REGION Network 86: Reset AI_PLC1_Loi_Truyen_Thong từ nút vật lý
   RUNG wire#powerrail
      Contact( "AI_Nut_Reset_Eff" )
      I_Contact( "AI_PLC1_EStop_Latch" )
      I_Contact( "AI_Nut_EStop_Eff" )
      R_Coil( "AI_PLC1_Loi_Truyen_Thong" )
   END_RUNG
   // the same network as SCL:
   IF "AI_Nut_Reset_Eff" AND NOT "AI_PLC1_EStop_Latch" AND NOT "AI_Nut_EStop_Eff" THEN
       "AI_PLC1_Loi_Truyen_Thong" := FALSE;
   END_IF;
END_REGION

REGION Network 87: Reset AI_PID_Bon2_Error từ nút vật lý
   RUNG wire#powerrail
      Contact( "AI_Nut_Reset_Eff" )
      I_Contact( "AI_PLC1_EStop_Latch" )
      I_Contact( "AI_Nut_EStop_Eff" )
      R_Coil( "AI_PID_Bon2_Error" )
   END_RUNG
   // the same network as SCL:
   IF "AI_Nut_Reset_Eff" AND NOT "AI_PLC1_EStop_Latch" AND NOT "AI_Nut_EStop_Eff" THEN
       "AI_PID_Bon2_Error" := FALSE;
   END_IF;
END_REGION

REGION Network 88: Reset AI_PLC1_Loi_Setpoint từ nút vật lý
   RUNG wire#powerrail
      Contact( "AI_Nut_Reset_Eff" )
      I_Contact( "AI_PLC1_EStop_Latch" )
      I_Contact( "AI_Nut_EStop_Eff" )
      R_Coil( "AI_PLC1_Loi_Setpoint" )
   END_RUNG
   // the same network as SCL:
   IF "AI_Nut_Reset_Eff" AND NOT "AI_PLC1_EStop_Latch" AND NOT "AI_Nut_EStop_Eff" THEN
       "AI_PLC1_Loi_Setpoint" := FALSE;
   END_IF;
END_REGION

REGION Network 89: Reset AI_BonChua_Loi_Setpoint từ nút vật lý
   RUNG wire#powerrail
      Contact( "AI_Nut_Reset_Eff" )
      I_Contact( "AI_PLC1_EStop_Latch" )
      I_Contact( "AI_Nut_EStop_Eff" )
      R_Coil( "AI_BonChua_Loi_Setpoint" )
   END_RUNG
   // the same network as SCL:
   IF "AI_Nut_Reset_Eff" AND NOT "AI_PLC1_EStop_Latch" AND NOT "AI_Nut_EStop_Eff" THEN
       "AI_BonChua_Loi_Setpoint" := FALSE;
   END_IF;
END_REGION

REGION Network 90: Reset AI_PLC1_Loi_Tong từ HMI
   RUNG wire#powerrail
      Contact( "AI_HMI_Reset_Alarm" )
      Contact( "AI_HMI_Cho_Phep_Sua_Thong_So" )
      I_Contact( "AI_PLC1_EStop_Latch" )
      I_Contact( "AI_Nut_EStop_Eff" )
      R_Coil( "AI_PLC1_Loi_Tong" )
   END_RUNG
   // the same network as SCL:
   IF "AI_HMI_Reset_Alarm" AND "AI_HMI_Cho_Phep_Sua_Thong_So" AND NOT "AI_PLC1_EStop_Latch" AND NOT "AI_Nut_EStop_Eff" THEN
       "AI_PLC1_Loi_Tong" := FALSE;
   END_IF;
END_REGION

REGION Network 91: Reset AI_PLC1_Loi_Dry_Run từ HMI
   RUNG wire#powerrail
      Contact( "AI_HMI_Reset_Alarm" )
      Contact( "AI_HMI_Cho_Phep_Sua_Thong_So" )
      I_Contact( "AI_PLC1_EStop_Latch" )
      I_Contact( "AI_Nut_EStop_Eff" )
      R_Coil( "AI_PLC1_Loi_Dry_Run" )
   END_RUNG
   // the same network as SCL:
   IF "AI_HMI_Reset_Alarm" AND "AI_HMI_Cho_Phep_Sua_Thong_So" AND NOT "AI_PLC1_EStop_Latch" AND NOT "AI_Nut_EStop_Eff" THEN
       "AI_PLC1_Loi_Dry_Run" := FALSE;
   END_IF;
END_REGION

REGION Network 92: Reset AI_PLC1_Loi_Dosing từ HMI
   RUNG wire#powerrail
      Contact( "AI_HMI_Reset_Alarm" )
      Contact( "AI_HMI_Cho_Phep_Sua_Thong_So" )
      I_Contact( "AI_PLC1_EStop_Latch" )
      I_Contact( "AI_Nut_EStop_Eff" )
      R_Coil( "AI_PLC1_Loi_Dosing" )
   END_RUNG
   // the same network as SCL:
   IF "AI_HMI_Reset_Alarm" AND "AI_HMI_Cho_Phep_Sua_Thong_So" AND NOT "AI_PLC1_EStop_Latch" AND NOT "AI_Nut_EStop_Eff" THEN
       "AI_PLC1_Loi_Dosing" := FALSE;
   END_IF;
END_REGION

REGION Network 93: Reset AI_PLC1_Loi_Truyen_Thong từ HMI
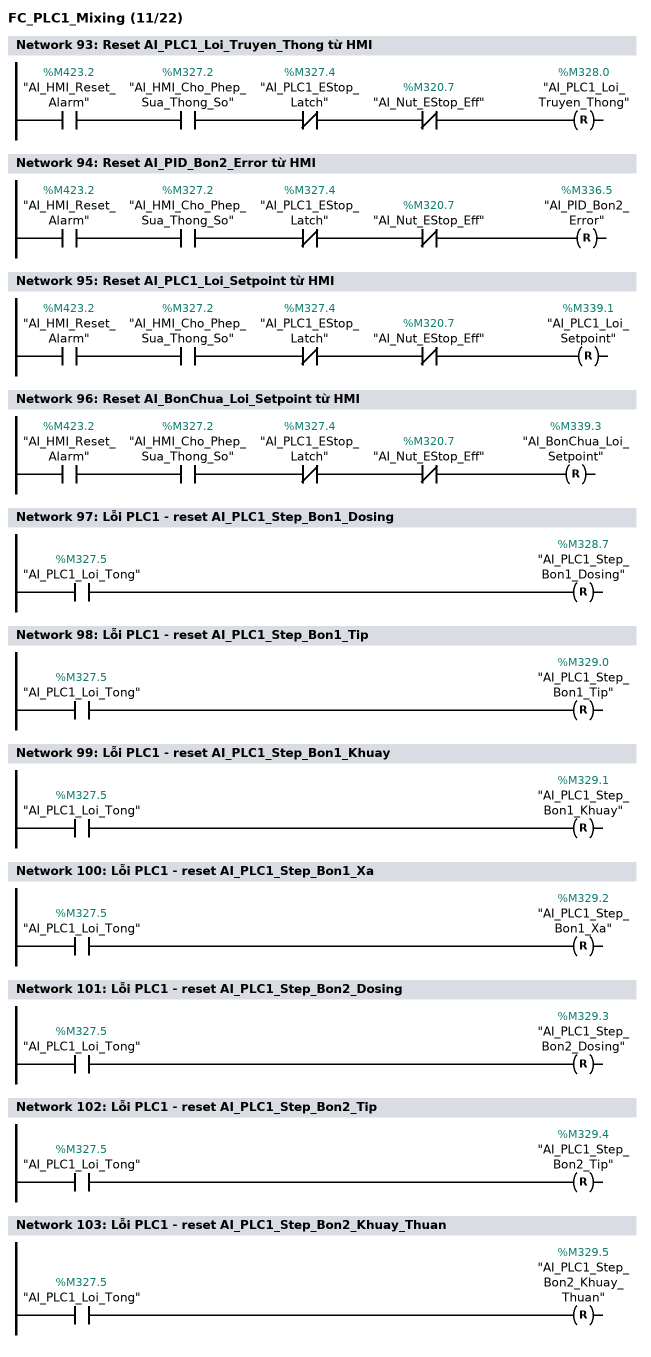
   RUNG wire#powerrail
      Contact( "AI_HMI_Reset_Alarm" )
      Contact( "AI_HMI_Cho_Phep_Sua_Thong_So" )
      I_Contact( "AI_PLC1_EStop_Latch" )
      I_Contact( "AI_Nut_EStop_Eff" )
      R_Coil( "AI_PLC1_Loi_Truyen_Thong" )
   END_RUNG
   // the same network as SCL:
   IF "AI_HMI_Reset_Alarm" AND "AI_HMI_Cho_Phep_Sua_Thong_So" AND NOT "AI_PLC1_EStop_Latch" AND NOT "AI_Nut_EStop_Eff" THEN
       "AI_PLC1_Loi_Truyen_Thong" := FALSE;
   END_IF;
END_REGION

REGION Network 94: Reset AI_PID_Bon2_Error từ HMI
   RUNG wire#powerrail
      Contact( "AI_HMI_Reset_Alarm" )
      Contact( "AI_HMI_Cho_Phep_Sua_Thong_So" )
      I_Contact( "AI_PLC1_EStop_Latch" )
      I_Contact( "AI_Nut_EStop_Eff" )
      R_Coil( "AI_PID_Bon2_Error" )
   END_RUNG
   // the same network as SCL:
   IF "AI_HMI_Reset_Alarm" AND "AI_HMI_Cho_Phep_Sua_Thong_So" AND NOT "AI_PLC1_EStop_Latch" AND NOT "AI_Nut_EStop_Eff" THEN
       "AI_PID_Bon2_Error" := FALSE;
   END_IF;
END_REGION

REGION Network 95: Reset AI_PLC1_Loi_Setpoint từ HMI
   RUNG wire#powerrail
      Contact( "AI_HMI_Reset_Alarm" )
      Contact( "AI_HMI_Cho_Phep_Sua_Thong_So" )
      I_Contact( "AI_PLC1_EStop_Latch" )
      I_Contact( "AI_Nut_EStop_Eff" )
      R_Coil( "AI_PLC1_Loi_Setpoint" )
   END_RUNG
   // the same network as SCL:
   IF "AI_HMI_Reset_Alarm" AND "AI_HMI_Cho_Phep_Sua_Thong_So" AND NOT "AI_PLC1_EStop_Latch" AND NOT "AI_Nut_EStop_Eff" THEN
       "AI_PLC1_Loi_Setpoint" := FALSE;
   END_IF;
END_REGION

REGION Network 96: Reset AI_BonChua_Loi_Setpoint từ HMI
   RUNG wire#powerrail
      Contact( "AI_HMI_Reset_Alarm" )
      Contact( "AI_HMI_Cho_Phep_Sua_Thong_So" )
      I_Contact( "AI_PLC1_EStop_Latch" )
      I_Contact( "AI_Nut_EStop_Eff" )
      R_Coil( "AI_BonChua_Loi_Setpoint" )
   END_RUNG
   // the same network as SCL:
   IF "AI_HMI_Reset_Alarm" AND "AI_HMI_Cho_Phep_Sua_Thong_So" AND NOT "AI_PLC1_EStop_Latch" AND NOT "AI_Nut_EStop_Eff" THEN
       "AI_BonChua_Loi_Setpoint" := FALSE;
   END_IF;
END_REGION

REGION Network 97: Lỗi PLC1 - reset AI_PLC1_Step_Bon1_Dosing
   RUNG wire#powerrail
      Contact( "AI_PLC1_Loi_Tong" )
      R_Coil( "AI_PLC1_Step_Bon1_Dosing" )
   END_RUNG
   // the same network as SCL:
   IF "AI_PLC1_Loi_Tong" THEN "AI_PLC1_Step_Bon1_Dosing" := FALSE; END_IF;
END_REGION

REGION Network 98: Lỗi PLC1 - reset AI_PLC1_Step_Bon1_Tip
   RUNG wire#powerrail
      Contact( "AI_PLC1_Loi_Tong" )
      R_Coil( "AI_PLC1_Step_Bon1_Tip" )
   END_RUNG
   // the same network as SCL:
   IF "AI_PLC1_Loi_Tong" THEN "AI_PLC1_Step_Bon1_Tip" := FALSE; END_IF;
END_REGION

REGION Network 99: Lỗi PLC1 - reset AI_PLC1_Step_Bon1_Khuay
   RUNG wire#powerrail
      Contact( "AI_PLC1_Loi_Tong" )
      R_Coil( "AI_PLC1_Step_Bon1_Khuay" )
   END_RUNG
   // the same network as SCL:
   IF "AI_PLC1_Loi_Tong" THEN "AI_PLC1_Step_Bon1_Khuay" := FALSE; END_IF;
END_REGION

REGION Network 100: Lỗi PLC1 - reset AI_PLC1_Step_Bon1_Xa
   RUNG wire#powerrail
      Contact( "AI_PLC1_Loi_Tong" )
      R_Coil( "AI_PLC1_Step_Bon1_Xa" )
   END_RUNG
   // the same network as SCL:
   IF "AI_PLC1_Loi_Tong" THEN "AI_PLC1_Step_Bon1_Xa" := FALSE; END_IF;
END_REGION

REGION Network 101: Lỗi PLC1 - reset AI_PLC1_Step_Bon2_Dosing
   RUNG wire#powerrail
      Contact( "AI_PLC1_Loi_Tong" )
      R_Coil( "AI_PLC1_Step_Bon2_Dosing" )
   END_RUNG
   // the same network as SCL:
   IF "AI_PLC1_Loi_Tong" THEN "AI_PLC1_Step_Bon2_Dosing" := FALSE; END_IF;
END_REGION

REGION Network 102: Lỗi PLC1 - reset AI_PLC1_Step_Bon2_Tip
   RUNG wire#powerrail
      Contact( "AI_PLC1_Loi_Tong" )
      R_Coil( "AI_PLC1_Step_Bon2_Tip" )
   END_RUNG
   // the same network as SCL:
   IF "AI_PLC1_Loi_Tong" THEN "AI_PLC1_Step_Bon2_Tip" := FALSE; END_IF;
END_REGION

REGION Network 103: Lỗi PLC1 - reset AI_PLC1_Step_Bon2_Khuay_Thuan
   RUNG wire#powerrail
      Contact( "AI_PLC1_Loi_Tong" )
      R_Coil( "AI_PLC1_Step_Bon2_Khuay_Thuan" )
   END_RUNG
   // the same network as SCL:
   IF "AI_PLC1_Loi_Tong" THEN "AI_PLC1_Step_Bon2_Khuay_Thuan" := FALSE; END_IF;
END_REGION

REGION Network 104: Lỗi PLC1 - reset AI_PLC1_Step_Bon2_Khuay_Nghich
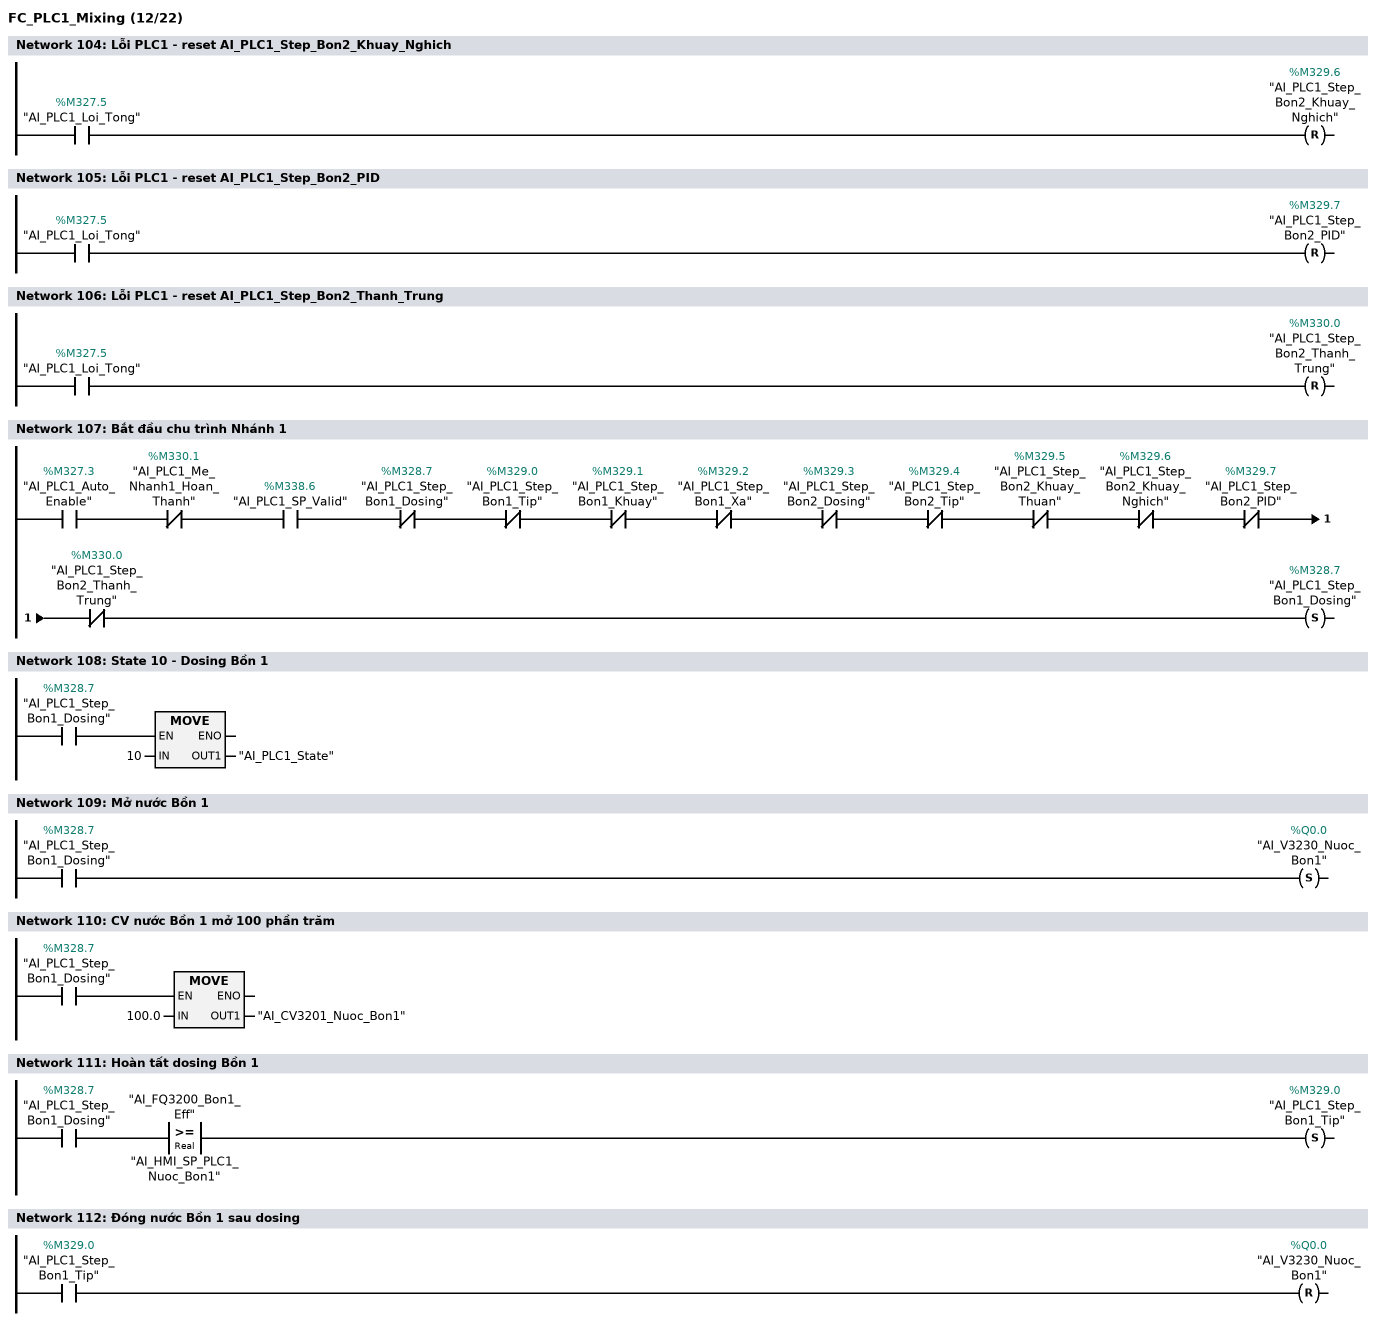
   RUNG wire#powerrail
      Contact( "AI_PLC1_Loi_Tong" )
      R_Coil( "AI_PLC1_Step_Bon2_Khuay_Nghich" )
   END_RUNG
   // the same network as SCL:
   IF "AI_PLC1_Loi_Tong" THEN "AI_PLC1_Step_Bon2_Khuay_Nghich" := FALSE; END_IF;
END_REGION

REGION Network 105: Lỗi PLC1 - reset AI_PLC1_Step_Bon2_PID
   RUNG wire#powerrail
      Contact( "AI_PLC1_Loi_Tong" )
      R_Coil( "AI_PLC1_Step_Bon2_PID" )
   END_RUNG
   // the same network as SCL:
   IF "AI_PLC1_Loi_Tong" THEN "AI_PLC1_Step_Bon2_PID" := FALSE; END_IF;
END_REGION

REGION Network 106: Lỗi PLC1 - reset AI_PLC1_Step_Bon2_Thanh_Trung
   RUNG wire#powerrail
      Contact( "AI_PLC1_Loi_Tong" )
      R_Coil( "AI_PLC1_Step_Bon2_Thanh_Trung" )
   END_RUNG
   // the same network as SCL:
   IF "AI_PLC1_Loi_Tong" THEN "AI_PLC1_Step_Bon2_Thanh_Trung" := FALSE; END_IF;
END_REGION

REGION Network 107: Bắt đầu chu trình Nhánh 1
   RUNG wire#powerrail
      Contact( "AI_PLC1_Auto_Enable" )
      I_Contact( "AI_PLC1_Me_Nhanh1_Hoan_Thanh" )
      Contact( "AI_PLC1_SP_Valid" )
      I_Contact( "AI_PLC1_Step_Bon1_Dosing" )
      I_Contact( "AI_PLC1_Step_Bon1_Tip" )
      I_Contact( "AI_PLC1_Step_Bon1_Khuay" )
      I_Contact( "AI_PLC1_Step_Bon1_Xa" )
      I_Contact( "AI_PLC1_Step_Bon2_Dosing" )
      I_Contact( "AI_PLC1_Step_Bon2_Tip" )
      I_Contact( "AI_PLC1_Step_Bon2_Khuay_Thuan" )
      I_Contact( "AI_PLC1_Step_Bon2_Khuay_Nghich" )
      I_Contact( "AI_PLC1_Step_Bon2_PID" )
      I_Contact( "AI_PLC1_Step_Bon2_Thanh_Trung" )
      S_Coil( "AI_PLC1_Step_Bon1_Dosing" )
   END_RUNG
   // the same network as SCL:
   IF "AI_PLC1_Auto_Enable" AND NOT "AI_PLC1_Me_Nhanh1_Hoan_Thanh" AND "AI_PLC1_SP_Valid" AND NOT "AI_PLC1_Step_Bon1_Dosing" AND NOT "AI_PLC1_Step_Bon1_Tip" AND NOT "AI_PLC1_Step_Bon1_Khuay" AND NOT "AI_PLC1_Step_Bon1_Xa" AND NOT "AI_PLC1_Step_Bon2_Dosing" AND NOT "AI_PLC1_Step_Bon2_Tip" AND NOT "AI_PLC1_Step_Bon2_Khuay_Thuan" AND NOT "AI_PLC1_Step_Bon2_Khuay_Nghich" AND NOT "AI_PLC1_Step_Bon2_PID" AND NOT "AI_PLC1_Step_Bon2_Thanh_Trung" THEN
       "AI_PLC1_Step_Bon1_Dosing" := TRUE;
   END_IF;
END_REGION

REGION Network 108: State 10 - Dosing Bồn 1
   RUNG wire#powerrail
      Contact( "AI_PLC1_Step_Bon1_Dosing" )
      { S7_GenerateENO := "TRUE" } Move(in := 10, out1 => "AI_PLC1_State")
   END_RUNG
   // the same network as SCL:
   IF "AI_PLC1_Step_Bon1_Dosing" THEN "AI_PLC1_State" := 10; END_IF;
END_REGION

REGION Network 109: Mở nước Bồn 1
   RUNG wire#powerrail
      Contact( "AI_PLC1_Step_Bon1_Dosing" )
      S_Coil( "AI_V3230_Nuoc_Bon1" )
   END_RUNG
   // the same network as SCL:
   IF "AI_PLC1_Step_Bon1_Dosing" THEN "AI_V3230_Nuoc_Bon1" := TRUE; END_IF;
END_REGION

REGION Network 110: CV nước Bồn 1 mở 100 phần trăm
   RUNG wire#powerrail
      Contact( "AI_PLC1_Step_Bon1_Dosing" )
      { S7_GenerateENO := "TRUE" } Move(in := 100.0, out1 => "AI_CV3201_Nuoc_Bon1")
   END_RUNG
   // the same network as SCL:
   IF "AI_PLC1_Step_Bon1_Dosing" THEN "AI_CV3201_Nuoc_Bon1" := 100.0; END_IF;
END_REGION

REGION Network 111: Hoàn tất dosing Bồn 1
   RUNG wire#powerrail
      Contact( "AI_PLC1_Step_Bon1_Dosing" )
      { S7_Templates := "SrcType := Real" } GE_Contact(in1 := "AI_FQ3200_Bon1_Eff", in2 := "AI_HMI_SP_PLC1_Nuoc_Bon1")
      S_Coil( "AI_PLC1_Step_Bon1_Tip" )
   END_RUNG
   // the same network as SCL:
   IF "AI_PLC1_Step_Bon1_Dosing" AND ("AI_FQ3200_Bon1_Eff" >= "AI_HMI_SP_PLC1_Nuoc_Bon1") THEN
       "AI_PLC1_Step_Bon1_Tip" := TRUE;
   END_IF;
END_REGION

REGION Network 112: Đóng nước Bồn 1 sau dosing
   RUNG wire#powerrail
      Contact( "AI_PLC1_Step_Bon1_Tip" )
      R_Coil( "AI_V3230_Nuoc_Bon1" )
   END_RUNG
   // the same network as SCL:
   IF "AI_PLC1_Step_Bon1_Tip" THEN "AI_V3230_Nuoc_Bon1" := FALSE; END_IF;
END_REGION

REGION Network 113: Reset bước dosing Bồn 1
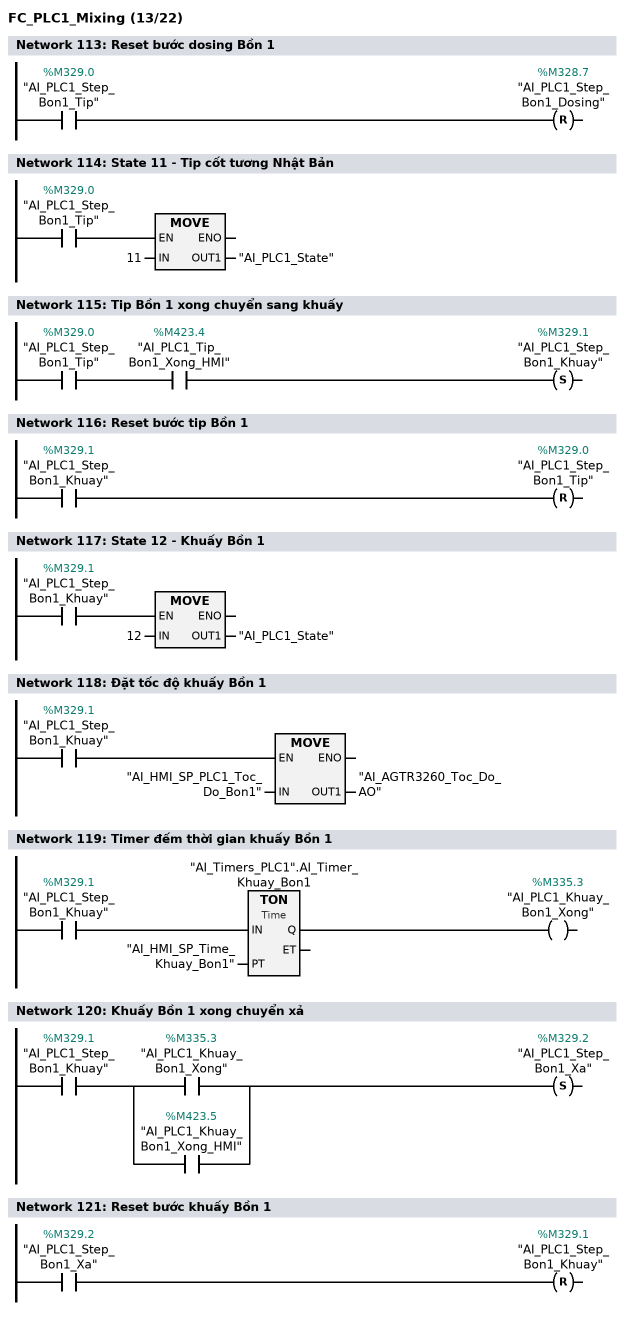
   RUNG wire#powerrail
      Contact( "AI_PLC1_Step_Bon1_Tip" )
      R_Coil( "AI_PLC1_Step_Bon1_Dosing" )
   END_RUNG
   // the same network as SCL:
   IF "AI_PLC1_Step_Bon1_Tip" THEN "AI_PLC1_Step_Bon1_Dosing" := FALSE; END_IF;
END_REGION

REGION Network 114: State 11 - Tip cốt tương Nhật Bản
   RUNG wire#powerrail
      Contact( "AI_PLC1_Step_Bon1_Tip" )
      { S7_GenerateENO := "TRUE" } Move(in := 11, out1 => "AI_PLC1_State")
   END_RUNG
   // the same network as SCL:
   IF "AI_PLC1_Step_Bon1_Tip" THEN "AI_PLC1_State" := 11; END_IF;
END_REGION

REGION Network 115: Tip Bồn 1 xong chuyển sang khuấy
   RUNG wire#powerrail
      Contact( "AI_PLC1_Step_Bon1_Tip" )
      Contact( "AI_PLC1_Tip_Bon1_Xong_HMI" )
      S_Coil( "AI_PLC1_Step_Bon1_Khuay" )
   END_RUNG
   // the same network as SCL:
   IF "AI_PLC1_Step_Bon1_Tip" AND "AI_PLC1_Tip_Bon1_Xong_HMI" THEN "AI_PLC1_Step_Bon1_Khuay" := TRUE; END_IF;
END_REGION

REGION Network 116: Reset bước tip Bồn 1
   RUNG wire#powerrail
      Contact( "AI_PLC1_Step_Bon1_Khuay" )
      R_Coil( "AI_PLC1_Step_Bon1_Tip" )
   END_RUNG
   // the same network as SCL:
   IF "AI_PLC1_Step_Bon1_Khuay" THEN "AI_PLC1_Step_Bon1_Tip" := FALSE; END_IF;
END_REGION

REGION Network 117: State 12 - Khuấy Bồn 1
   RUNG wire#powerrail
      Contact( "AI_PLC1_Step_Bon1_Khuay" )
      { S7_GenerateENO := "TRUE" } Move(in := 12, out1 => "AI_PLC1_State")
   END_RUNG
   // the same network as SCL:
   IF "AI_PLC1_Step_Bon1_Khuay" THEN "AI_PLC1_State" := 12; END_IF;
END_REGION

REGION Network 118: Đặt tốc độ khuấy Bồn 1
   RUNG wire#powerrail
      Contact( "AI_PLC1_Step_Bon1_Khuay" )
      { S7_GenerateENO := "TRUE" } Move(in := "AI_HMI_SP_PLC1_Toc_Do_Bon1", out1 => "AI_AGTR3260_Toc_Do_AO")
   END_RUNG
   // the same network as SCL:
   IF "AI_PLC1_Step_Bon1_Khuay" THEN "AI_AGTR3260_Toc_Do_AO" := "AI_HMI_SP_PLC1_Toc_Do_Bon1"; END_IF;
END_REGION

REGION Network 119: Timer đếm thời gian khuấy Bồn 1
   RUNG wire#powerrail
      Contact( "AI_PLC1_Step_Bon1_Khuay" )
      { S7_Templates := "time_type := Time" } "AI_Timers_PLC1".AI_Timer_Khuay_Bon1.TON(pt := "AI_HMI_SP_Time_Khuay_Bon1", et =>)
      Coil( "AI_PLC1_Khuay_Bon1_Xong" )
   END_RUNG
   // the same network as SCL:
   "AI_Timers_PLC1".AI_Timer_Khuay_Bon1.TON(IN := "AI_PLC1_Step_Bon1_Khuay", PT := "AI_HMI_SP_Time_Khuay_Bon1");
   "AI_PLC1_Khuay_Bon1_Xong" := "AI_Timers_PLC1".AI_Timer_Khuay_Bon1.Q;
END_REGION

REGION Network 120: Khuấy Bồn 1 xong chuyển xả
   RUNG wire#powerrail
      Contact( "AI_PLC1_Step_Bon1_Khuay" )
      wire#w1
      Contact( "AI_PLC1_Khuay_Bon1_Xong" )
      wire#w2
      S_Coil( "AI_PLC1_Step_Bon1_Xa" )
   END_RUNG
   RUNG wire#w1
      Contact( "AI_PLC1_Khuay_Bon1_Xong_HMI" )
   END_RUNG wire#w2
   // the same network as SCL:
   IF "AI_PLC1_Step_Bon1_Khuay" AND ("AI_PLC1_Khuay_Bon1_Xong" OR "AI_PLC1_Khuay_Bon1_Xong_HMI") THEN
       "AI_PLC1_Step_Bon1_Xa" := TRUE;
   END_IF;
END_REGION

REGION Network 121: Reset bước khuấy Bồn 1
   RUNG wire#powerrail
      Contact( "AI_PLC1_Step_Bon1_Xa" )
      R_Coil( "AI_PLC1_Step_Bon1_Khuay" )
   END_RUNG
   // the same network as SCL:
   IF "AI_PLC1_Step_Bon1_Xa" THEN "AI_PLC1_Step_Bon1_Khuay" := FALSE; END_IF;
END_REGION

REGION Network 122: State 15 - Xả Bồn 1 sang Bồn 2
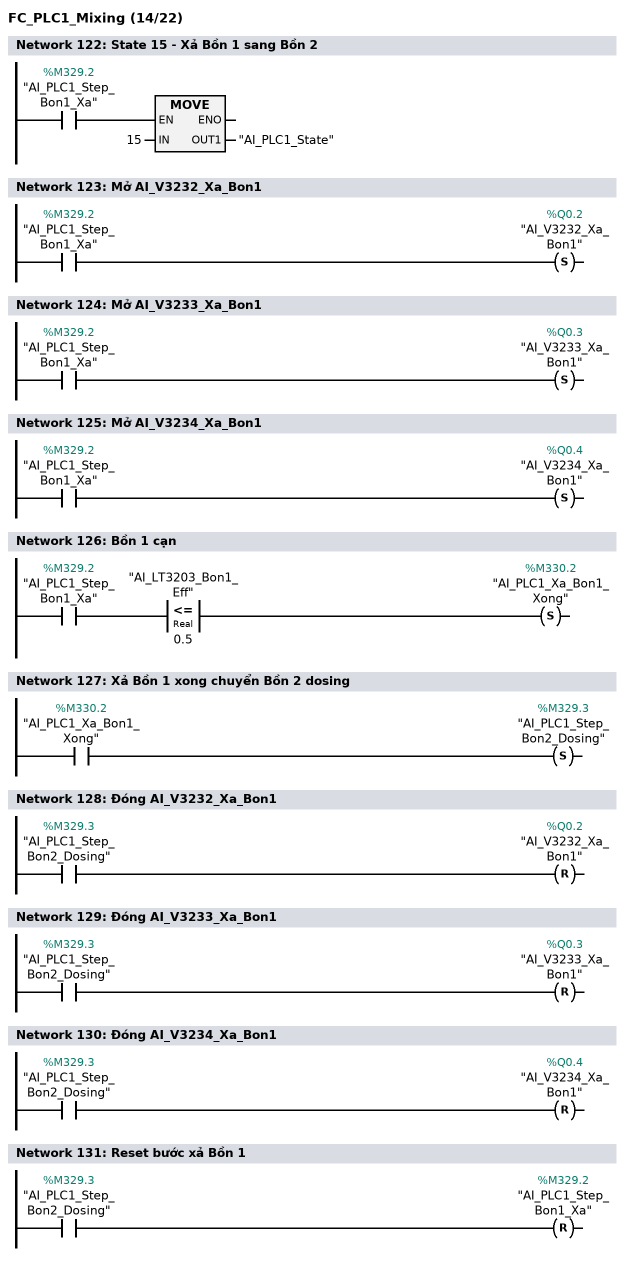
   RUNG wire#powerrail
      Contact( "AI_PLC1_Step_Bon1_Xa" )
      { S7_GenerateENO := "TRUE" } Move(in := 15, out1 => "AI_PLC1_State")
   END_RUNG
   // the same network as SCL:
   IF "AI_PLC1_Step_Bon1_Xa" THEN "AI_PLC1_State" := 15; END_IF;
END_REGION

REGION Network 123: Mở AI_V3232_Xa_Bon1
   RUNG wire#powerrail
      Contact( "AI_PLC1_Step_Bon1_Xa" )
      S_Coil( "AI_V3232_Xa_Bon1" )
   END_RUNG
   // the same network as SCL:
   IF "AI_PLC1_Step_Bon1_Xa" THEN "AI_V3232_Xa_Bon1" := TRUE; END_IF;
END_REGION

REGION Network 124: Mở AI_V3233_Xa_Bon1
   RUNG wire#powerrail
      Contact( "AI_PLC1_Step_Bon1_Xa" )
      S_Coil( "AI_V3233_Xa_Bon1" )
   END_RUNG
   // the same network as SCL:
   IF "AI_PLC1_Step_Bon1_Xa" THEN "AI_V3233_Xa_Bon1" := TRUE; END_IF;
END_REGION

REGION Network 125: Mở AI_V3234_Xa_Bon1
   RUNG wire#powerrail
      Contact( "AI_PLC1_Step_Bon1_Xa" )
      S_Coil( "AI_V3234_Xa_Bon1" )
   END_RUNG
   // the same network as SCL:
   IF "AI_PLC1_Step_Bon1_Xa" THEN "AI_V3234_Xa_Bon1" := TRUE; END_IF;
END_REGION

REGION Network 126: Bồn 1 cạn
   RUNG wire#powerrail
      Contact( "AI_PLC1_Step_Bon1_Xa" )
      { S7_Templates := "SrcType := Real" } LE_Contact(in1 := "AI_LT3203_Bon1_Eff", in2 := 0.5)
      S_Coil( "AI_PLC1_Xa_Bon1_Xong" )
   END_RUNG
   // the same network as SCL:
   IF "AI_PLC1_Step_Bon1_Xa" AND ("AI_LT3203_Bon1_Eff" <= 0.5) THEN "AI_PLC1_Xa_Bon1_Xong" := TRUE; END_IF;
END_REGION

REGION Network 127: Xả Bồn 1 xong chuyển Bồn 2 dosing
   RUNG wire#powerrail
      Contact( "AI_PLC1_Xa_Bon1_Xong" )
      S_Coil( "AI_PLC1_Step_Bon2_Dosing" )
   END_RUNG
   // the same network as SCL:
   IF "AI_PLC1_Xa_Bon1_Xong" THEN "AI_PLC1_Step_Bon2_Dosing" := TRUE; END_IF;
END_REGION

REGION Network 128: Đóng AI_V3232_Xa_Bon1
   RUNG wire#powerrail
      Contact( "AI_PLC1_Step_Bon2_Dosing" )
      R_Coil( "AI_V3232_Xa_Bon1" )
   END_RUNG
   // the same network as SCL:
   IF "AI_PLC1_Step_Bon2_Dosing" THEN "AI_V3232_Xa_Bon1" := FALSE; END_IF;
END_REGION

REGION Network 129: Đóng AI_V3233_Xa_Bon1
   RUNG wire#powerrail
      Contact( "AI_PLC1_Step_Bon2_Dosing" )
      R_Coil( "AI_V3233_Xa_Bon1" )
   END_RUNG
   // the same network as SCL:
   IF "AI_PLC1_Step_Bon2_Dosing" THEN "AI_V3233_Xa_Bon1" := FALSE; END_IF;
END_REGION

REGION Network 130: Đóng AI_V3234_Xa_Bon1
   RUNG wire#powerrail
      Contact( "AI_PLC1_Step_Bon2_Dosing" )
      R_Coil( "AI_V3234_Xa_Bon1" )
   END_RUNG
   // the same network as SCL:
   IF "AI_PLC1_Step_Bon2_Dosing" THEN "AI_V3234_Xa_Bon1" := FALSE; END_IF;
END_REGION

REGION Network 131: Reset bước xả Bồn 1
   RUNG wire#powerrail
      Contact( "AI_PLC1_Step_Bon2_Dosing" )
      R_Coil( "AI_PLC1_Step_Bon1_Xa" )
   END_RUNG
   // the same network as SCL:
   IF "AI_PLC1_Step_Bon2_Dosing" THEN "AI_PLC1_Step_Bon1_Xa" := FALSE; END_IF;
END_REGION

REGION Network 132: State 20 - Dosing Bồn 2
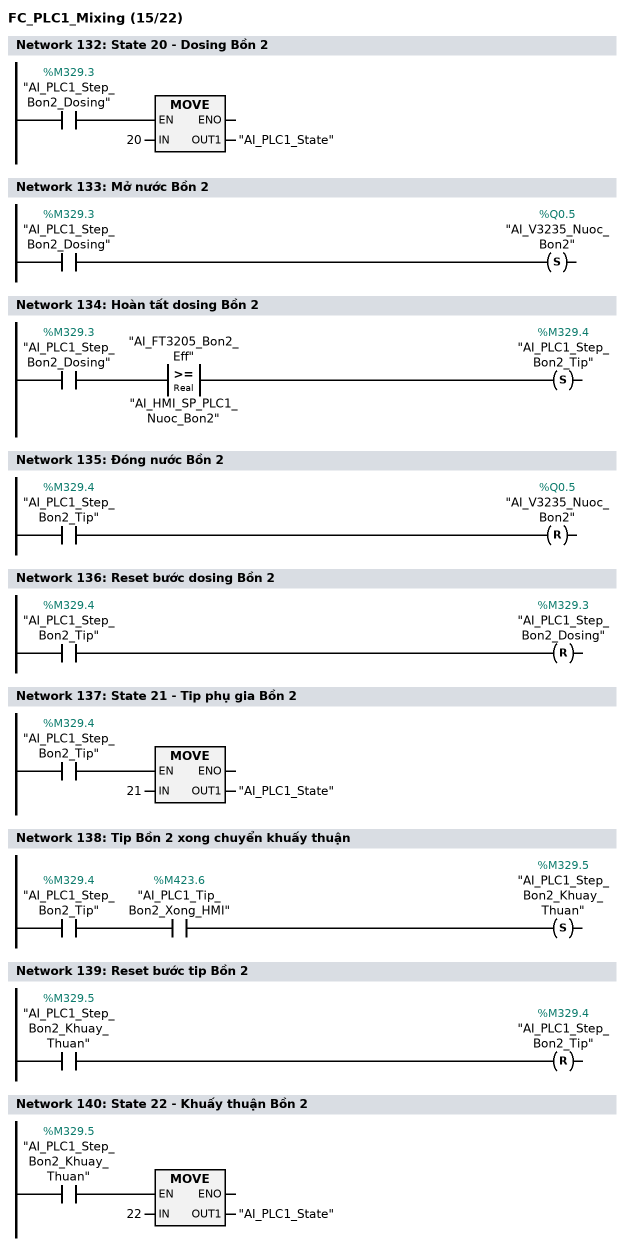
   RUNG wire#powerrail
      Contact( "AI_PLC1_Step_Bon2_Dosing" )
      { S7_GenerateENO := "TRUE" } Move(in := 20, out1 => "AI_PLC1_State")
   END_RUNG
   // the same network as SCL:
   IF "AI_PLC1_Step_Bon2_Dosing" THEN "AI_PLC1_State" := 20; END_IF;
END_REGION

REGION Network 133: Mở nước Bồn 2
   RUNG wire#powerrail
      Contact( "AI_PLC1_Step_Bon2_Dosing" )
      S_Coil( "AI_V3235_Nuoc_Bon2" )
   END_RUNG
   // the same network as SCL:
   IF "AI_PLC1_Step_Bon2_Dosing" THEN "AI_V3235_Nuoc_Bon2" := TRUE; END_IF;
END_REGION

REGION Network 134: Hoàn tất dosing Bồn 2
   RUNG wire#powerrail
      Contact( "AI_PLC1_Step_Bon2_Dosing" )
      { S7_Templates := "SrcType := Real" } GE_Contact(in1 := "AI_FT3205_Bon2_Eff", in2 := "AI_HMI_SP_PLC1_Nuoc_Bon2")
      S_Coil( "AI_PLC1_Step_Bon2_Tip" )
   END_RUNG
   // the same network as SCL:
   IF "AI_PLC1_Step_Bon2_Dosing" AND ("AI_FT3205_Bon2_Eff" >= "AI_HMI_SP_PLC1_Nuoc_Bon2") THEN
       "AI_PLC1_Step_Bon2_Tip" := TRUE;
   END_IF;
END_REGION

REGION Network 135: Đóng nước Bồn 2
   RUNG wire#powerrail
      Contact( "AI_PLC1_Step_Bon2_Tip" )
      R_Coil( "AI_V3235_Nuoc_Bon2" )
   END_RUNG
   // the same network as SCL:
   IF "AI_PLC1_Step_Bon2_Tip" THEN "AI_V3235_Nuoc_Bon2" := FALSE; END_IF;
END_REGION

REGION Network 136: Reset bước dosing Bồn 2
   RUNG wire#powerrail
      Contact( "AI_PLC1_Step_Bon2_Tip" )
      R_Coil( "AI_PLC1_Step_Bon2_Dosing" )
   END_RUNG
   // the same network as SCL:
   IF "AI_PLC1_Step_Bon2_Tip" THEN "AI_PLC1_Step_Bon2_Dosing" := FALSE; END_IF;
END_REGION

REGION Network 137: State 21 - Tip phụ gia Bồn 2
   RUNG wire#powerrail
      Contact( "AI_PLC1_Step_Bon2_Tip" )
      { S7_GenerateENO := "TRUE" } Move(in := 21, out1 => "AI_PLC1_State")
   END_RUNG
   // the same network as SCL:
   IF "AI_PLC1_Step_Bon2_Tip" THEN "AI_PLC1_State" := 21; END_IF;
END_REGION

REGION Network 138: Tip Bồn 2 xong chuyển khuấy thuận
   RUNG wire#powerrail
      Contact( "AI_PLC1_Step_Bon2_Tip" )
      Contact( "AI_PLC1_Tip_Bon2_Xong_HMI" )
      S_Coil( "AI_PLC1_Step_Bon2_Khuay_Thuan" )
   END_RUNG
   // the same network as SCL:
   IF "AI_PLC1_Step_Bon2_Tip" AND "AI_PLC1_Tip_Bon2_Xong_HMI" THEN
       "AI_PLC1_Step_Bon2_Khuay_Thuan" := TRUE;
   END_IF;
END_REGION

REGION Network 139: Reset bước tip Bồn 2
   RUNG wire#powerrail
      Contact( "AI_PLC1_Step_Bon2_Khuay_Thuan" )
      R_Coil( "AI_PLC1_Step_Bon2_Tip" )
   END_RUNG
   // the same network as SCL:
   IF "AI_PLC1_Step_Bon2_Khuay_Thuan" THEN "AI_PLC1_Step_Bon2_Tip" := FALSE; END_IF;
END_REGION

REGION Network 140: State 22 - Khuấy thuận Bồn 2
   RUNG wire#powerrail
      Contact( "AI_PLC1_Step_Bon2_Khuay_Thuan" )
      { S7_GenerateENO := "TRUE" } Move(in := 22, out1 => "AI_PLC1_State")
   END_RUNG
   // the same network as SCL:
   IF "AI_PLC1_Step_Bon2_Khuay_Thuan" THEN "AI_PLC1_State" := 22; END_IF;
END_REGION

REGION Network 141: Tốc độ khuấy thuận Bồn 2
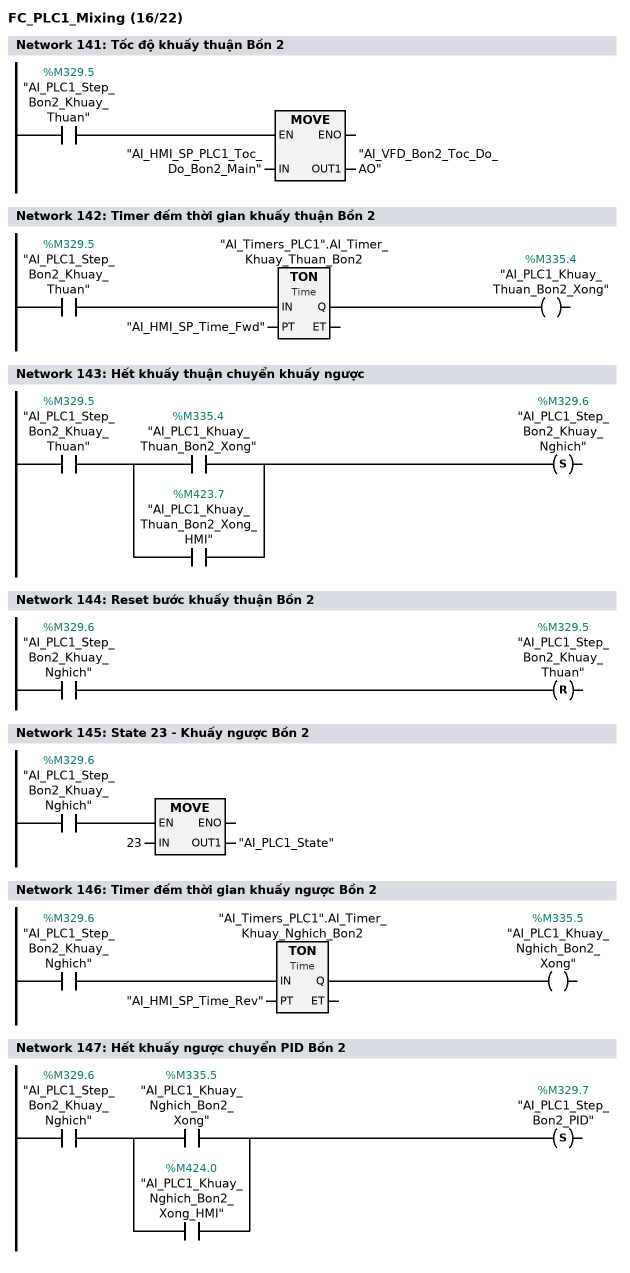
   RUNG wire#powerrail
      Contact( "AI_PLC1_Step_Bon2_Khuay_Thuan" )
      { S7_GenerateENO := "TRUE" } Move(in := "AI_HMI_SP_PLC1_Toc_Do_Bon2_Main", out1 => "AI_VFD_Bon2_Toc_Do_AO")
   END_RUNG
   // the same network as SCL:
   IF "AI_PLC1_Step_Bon2_Khuay_Thuan" THEN
       "AI_VFD_Bon2_Toc_Do_AO" := "AI_HMI_SP_PLC1_Toc_Do_Bon2_Main";
   END_IF;
END_REGION

REGION Network 142: Timer đếm thời gian khuấy thuận Bồn 2
   RUNG wire#powerrail
      Contact( "AI_PLC1_Step_Bon2_Khuay_Thuan" )
      { S7_Templates := "time_type := Time" } "AI_Timers_PLC1".AI_Timer_Khuay_Thuan_Bon2.TON(pt := "AI_HMI_SP_Time_Fwd", et =>)
      Coil( "AI_PLC1_Khuay_Thuan_Bon2_Xong" )
   END_RUNG
   // the same network as SCL:
   "AI_Timers_PLC1".AI_Timer_Khuay_Thuan_Bon2.TON(IN := "AI_PLC1_Step_Bon2_Khuay_Thuan",
                           PT := "AI_HMI_SP_Time_Fwd");
   "AI_PLC1_Khuay_Thuan_Bon2_Xong" := "AI_Timers_PLC1".AI_Timer_Khuay_Thuan_Bon2.Q;
END_REGION

REGION Network 143: Hết khuấy thuận chuyển khuấy ngược
   RUNG wire#powerrail
      Contact( "AI_PLC1_Step_Bon2_Khuay_Thuan" )
      wire#w1
      Contact( "AI_PLC1_Khuay_Thuan_Bon2_Xong" )
      wire#w2
      S_Coil( "AI_PLC1_Step_Bon2_Khuay_Nghich" )
   END_RUNG
   RUNG wire#w1
      Contact( "AI_PLC1_Khuay_Thuan_Bon2_Xong_HMI" )
   END_RUNG wire#w2
   // the same network as SCL:
   IF "AI_PLC1_Step_Bon2_Khuay_Thuan" AND ("AI_PLC1_Khuay_Thuan_Bon2_Xong" OR "AI_PLC1_Khuay_Thuan_Bon2_Xong_HMI") THEN
       "AI_PLC1_Step_Bon2_Khuay_Nghich" := TRUE;
   END_IF;
END_REGION

REGION Network 144: Reset bước khuấy thuận Bồn 2
   RUNG wire#powerrail
      Contact( "AI_PLC1_Step_Bon2_Khuay_Nghich" )
      R_Coil( "AI_PLC1_Step_Bon2_Khuay_Thuan" )
   END_RUNG
   // the same network as SCL:
   IF "AI_PLC1_Step_Bon2_Khuay_Nghich" THEN "AI_PLC1_Step_Bon2_Khuay_Thuan" := FALSE; END_IF;
END_REGION

REGION Network 145: State 23 - Khuấy ngược Bồn 2
   RUNG wire#powerrail
      Contact( "AI_PLC1_Step_Bon2_Khuay_Nghich" )
      { S7_GenerateENO := "TRUE" } Move(in := 23, out1 => "AI_PLC1_State")
   END_RUNG
   // the same network as SCL:
   IF "AI_PLC1_Step_Bon2_Khuay_Nghich" THEN "AI_PLC1_State" := 23; END_IF;
END_REGION

REGION Network 146: Timer đếm thời gian khuấy ngược Bồn 2
   RUNG wire#powerrail
      Contact( "AI_PLC1_Step_Bon2_Khuay_Nghich" )
      { S7_Templates := "time_type := Time" } "AI_Timers_PLC1".AI_Timer_Khuay_Nghich_Bon2.TON(pt := "AI_HMI_SP_Time_Rev", et =>)
      Coil( "AI_PLC1_Khuay_Nghich_Bon2_Xong" )
   END_RUNG
   // the same network as SCL:
   "AI_Timers_PLC1".AI_Timer_Khuay_Nghich_Bon2.TON(IN := "AI_PLC1_Step_Bon2_Khuay_Nghich",
                           PT := "AI_HMI_SP_Time_Rev");
   "AI_PLC1_Khuay_Nghich_Bon2_Xong" := "AI_Timers_PLC1".AI_Timer_Khuay_Nghich_Bon2.Q;
END_REGION

REGION Network 147: Hết khuấy ngược chuyển PID Bồn 2
   RUNG wire#powerrail
      Contact( "AI_PLC1_Step_Bon2_Khuay_Nghich" )
      wire#w1
      Contact( "AI_PLC1_Khuay_Nghich_Bon2_Xong" )
      wire#w2
      S_Coil( "AI_PLC1_Step_Bon2_PID" )
   END_RUNG
   RUNG wire#w1
      Contact( "AI_PLC1_Khuay_Nghich_Bon2_Xong_HMI" )
   END_RUNG wire#w2
   // the same network as SCL:
   IF "AI_PLC1_Step_Bon2_Khuay_Nghich" AND ("AI_PLC1_Khuay_Nghich_Bon2_Xong" OR "AI_PLC1_Khuay_Nghich_Bon2_Xong_HMI") THEN
       "AI_PLC1_Step_Bon2_PID" := TRUE;
   END_IF;
END_REGION

REGION Network 148: Reset bước khuấy ngược Bồn 2
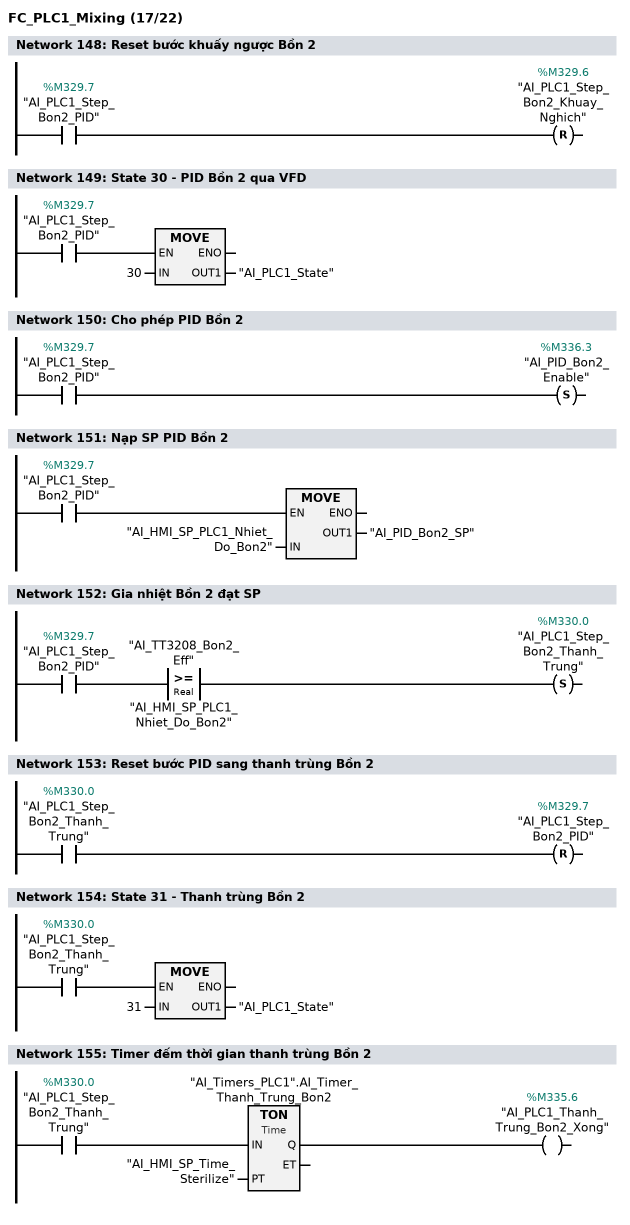
   RUNG wire#powerrail
      Contact( "AI_PLC1_Step_Bon2_PID" )
      R_Coil( "AI_PLC1_Step_Bon2_Khuay_Nghich" )
   END_RUNG
   // the same network as SCL:
   IF "AI_PLC1_Step_Bon2_PID" THEN "AI_PLC1_Step_Bon2_Khuay_Nghich" := FALSE; END_IF;
END_REGION

REGION Network 149: State 30 - PID Bồn 2 qua VFD
   RUNG wire#powerrail
      Contact( "AI_PLC1_Step_Bon2_PID" )
      { S7_GenerateENO := "TRUE" } Move(in := 30, out1 => "AI_PLC1_State")
   END_RUNG
   // the same network as SCL:
   IF "AI_PLC1_Step_Bon2_PID" THEN "AI_PLC1_State" := 30; END_IF;
END_REGION

REGION Network 150: Cho phép PID Bồn 2
   RUNG wire#powerrail
      Contact( "AI_PLC1_Step_Bon2_PID" )
      S_Coil( "AI_PID_Bon2_Enable" )
   END_RUNG
   // the same network as SCL:
   IF "AI_PLC1_Step_Bon2_PID" THEN "AI_PID_Bon2_Enable" := TRUE; END_IF;
END_REGION

REGION Network 151: Nạp SP PID Bồn 2
   RUNG wire#powerrail
      Contact( "AI_PLC1_Step_Bon2_PID" )
      { S7_GenerateENO := "TRUE" } Move(in := "AI_HMI_SP_PLC1_Nhiet_Do_Bon2", out1 => "AI_PID_Bon2_SP")
   END_RUNG
   // the same network as SCL:
   IF "AI_PLC1_Step_Bon2_PID" THEN "AI_PID_Bon2_SP" := "AI_HMI_SP_PLC1_Nhiet_Do_Bon2"; END_IF;
END_REGION

REGION Network 152: Gia nhiệt Bồn 2 đạt SP
   RUNG wire#powerrail
      Contact( "AI_PLC1_Step_Bon2_PID" )
      { S7_Templates := "SrcType := Real" } GE_Contact(in1 := "AI_TT3208_Bon2_Eff", in2 := "AI_HMI_SP_PLC1_Nhiet_Do_Bon2")
      S_Coil( "AI_PLC1_Step_Bon2_Thanh_Trung" )
   END_RUNG
   // the same network as SCL:
   IF "AI_PLC1_Step_Bon2_PID" AND ("AI_TT3208_Bon2_Eff" >= "AI_HMI_SP_PLC1_Nhiet_Do_Bon2") THEN
       "AI_PLC1_Step_Bon2_Thanh_Trung" := TRUE;
   END_IF;
END_REGION

REGION Network 153: Reset bước PID sang thanh trùng Bồn 2
   RUNG wire#powerrail
      Contact( "AI_PLC1_Step_Bon2_Thanh_Trung" )
      R_Coil( "AI_PLC1_Step_Bon2_PID" )
   END_RUNG
   // the same network as SCL:
   IF "AI_PLC1_Step_Bon2_Thanh_Trung" THEN "AI_PLC1_Step_Bon2_PID" := FALSE; END_IF;
END_REGION

REGION Network 154: State 31 - Thanh trùng Bồn 2
   RUNG wire#powerrail
      Contact( "AI_PLC1_Step_Bon2_Thanh_Trung" )
      { S7_GenerateENO := "TRUE" } Move(in := 31, out1 => "AI_PLC1_State")
   END_RUNG
   // the same network as SCL:
   IF "AI_PLC1_Step_Bon2_Thanh_Trung" THEN "AI_PLC1_State" := 31; END_IF;
END_REGION

REGION Network 155: Timer đếm thời gian thanh trùng Bồn 2
   RUNG wire#powerrail
      Contact( "AI_PLC1_Step_Bon2_Thanh_Trung" )
      { S7_Templates := "time_type := Time" } "AI_Timers_PLC1".AI_Timer_Thanh_Trung_Bon2.TON(pt := "AI_HMI_SP_Time_Sterilize", et =>)
      Coil( "AI_PLC1_Thanh_Trung_Bon2_Xong" )
   END_RUNG
   // the same network as SCL:
   "AI_Timers_PLC1".AI_Timer_Thanh_Trung_Bon2.TON(IN := "AI_PLC1_Step_Bon2_Thanh_Trung",
                           PT := "AI_HMI_SP_Time_Sterilize");
   "AI_PLC1_Thanh_Trung_Bon2_Xong" := "AI_Timers_PLC1".AI_Timer_Thanh_Trung_Bon2.Q;
END_REGION

REGION Network 156: Thanh trùng Bồn 2 xong
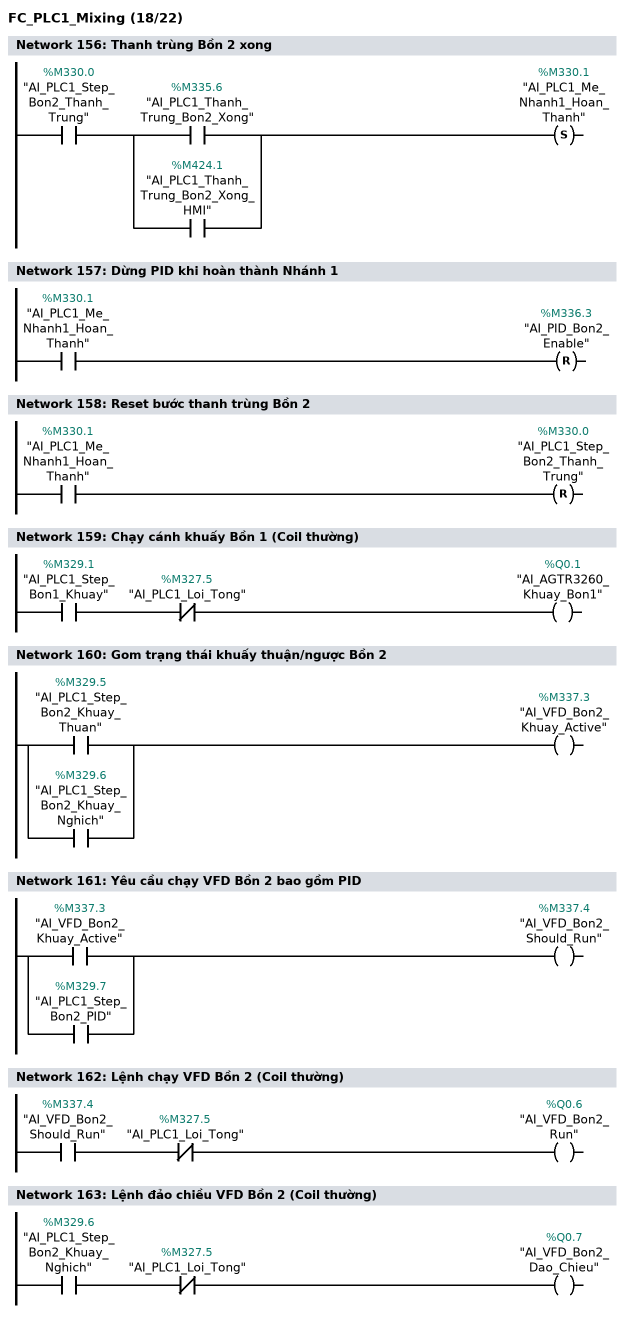
   RUNG wire#powerrail
      Contact( "AI_PLC1_Step_Bon2_Thanh_Trung" )
      wire#w1
      Contact( "AI_PLC1_Thanh_Trung_Bon2_Xong" )
      wire#w2
      S_Coil( "AI_PLC1_Me_Nhanh1_Hoan_Thanh" )
   END_RUNG
   RUNG wire#w1
      Contact( "AI_PLC1_Thanh_Trung_Bon2_Xong_HMI" )
   END_RUNG wire#w2
   // the same network as SCL:
   IF "AI_PLC1_Step_Bon2_Thanh_Trung" AND ("AI_PLC1_Thanh_Trung_Bon2_Xong" OR "AI_PLC1_Thanh_Trung_Bon2_Xong_HMI") THEN
       "AI_PLC1_Me_Nhanh1_Hoan_Thanh" := TRUE;
   END_IF;
END_REGION

REGION Network 157: Dừng PID khi hoàn thành Nhánh 1
   RUNG wire#powerrail
      Contact( "AI_PLC1_Me_Nhanh1_Hoan_Thanh" )
      R_Coil( "AI_PID_Bon2_Enable" )
   END_RUNG
   // the same network as SCL:
   IF "AI_PLC1_Me_Nhanh1_Hoan_Thanh" THEN "AI_PID_Bon2_Enable" := FALSE; END_IF;
END_REGION

REGION Network 158: Reset bước thanh trùng Bồn 2
   RUNG wire#powerrail
      Contact( "AI_PLC1_Me_Nhanh1_Hoan_Thanh" )
      R_Coil( "AI_PLC1_Step_Bon2_Thanh_Trung" )
   END_RUNG
   // the same network as SCL:
   IF "AI_PLC1_Me_Nhanh1_Hoan_Thanh" THEN "AI_PLC1_Step_Bon2_Thanh_Trung" := FALSE; END_IF;
END_REGION

REGION Network 159: Chạy cánh khuấy Bồn 1 (Coil thường)
   RUNG wire#powerrail
      Contact( "AI_PLC1_Step_Bon1_Khuay" )
      I_Contact( "AI_PLC1_Loi_Tong" )
      Coil( "AI_AGTR3260_Khuay_Bon1" )
   END_RUNG
   // the same network as SCL:
   "AI_AGTR3260_Khuay_Bon1" := "AI_PLC1_Step_Bon1_Khuay" AND NOT "AI_PLC1_Loi_Tong";
END_REGION

REGION Network 160: Gom trạng thái khuấy thuận/ngược Bồn 2
   RUNG wire#powerrail
      Contact( "AI_PLC1_Step_Bon2_Khuay_Thuan" )
      wire#w1
      Coil( "AI_VFD_Bon2_Khuay_Active" )
   END_RUNG
   RUNG wire#powerrail
      Contact( "AI_PLC1_Step_Bon2_Khuay_Nghich" )
   END_RUNG wire#w1
   // the same network as SCL:
   "AI_VFD_Bon2_Khuay_Active" := "AI_PLC1_Step_Bon2_Khuay_Thuan" OR "AI_PLC1_Step_Bon2_Khuay_Nghich";
END_REGION

REGION Network 161: Yêu cầu chạy VFD Bồn 2 bao gồm PID
   RUNG wire#powerrail
      Contact( "AI_VFD_Bon2_Khuay_Active" )
      wire#w1
      Coil( "AI_VFD_Bon2_Should_Run" )
   END_RUNG
   RUNG wire#powerrail
      Contact( "AI_PLC1_Step_Bon2_PID" )
   END_RUNG wire#w1
   // the same network as SCL:
   "AI_VFD_Bon2_Should_Run" := "AI_VFD_Bon2_Khuay_Active" OR "AI_PLC1_Step_Bon2_PID";
END_REGION

REGION Network 162: Lệnh chạy VFD Bồn 2 (Coil thường)
   RUNG wire#powerrail
      Contact( "AI_VFD_Bon2_Should_Run" )
      I_Contact( "AI_PLC1_Loi_Tong" )
      Coil( "AI_VFD_Bon2_Run" )
   END_RUNG
   // the same network as SCL:
   "AI_VFD_Bon2_Run" := "AI_VFD_Bon2_Should_Run" AND NOT "AI_PLC1_Loi_Tong";
END_REGION

REGION Network 163: Lệnh đảo chiều VFD Bồn 2 (Coil thường)
   RUNG wire#powerrail
      Contact( "AI_PLC1_Step_Bon2_Khuay_Nghich" )
      I_Contact( "AI_PLC1_Loi_Tong" )
      Coil( "AI_VFD_Bon2_Dao_Chieu" )
   END_RUNG
   // the same network as SCL:
   "AI_VFD_Bon2_Dao_Chieu" := "AI_PLC1_Step_Bon2_Khuay_Nghich" AND NOT "AI_PLC1_Loi_Tong";
END_REGION

REGION Network 164: Reset CV nước Bồn 1 khi không dosing
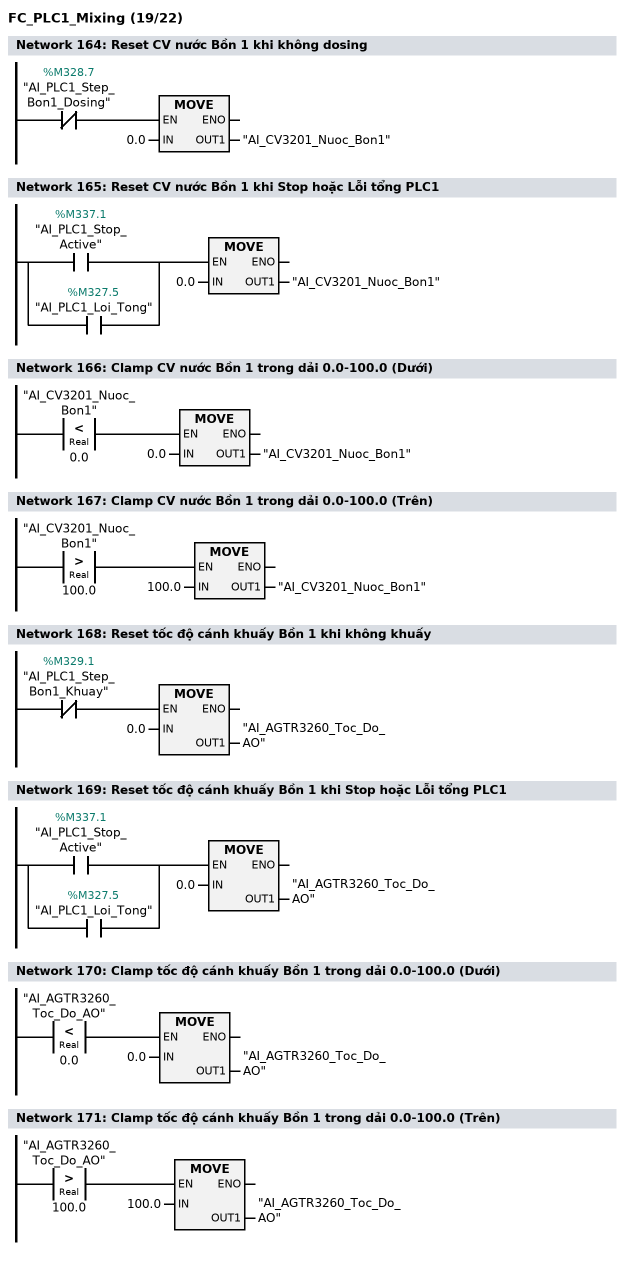
   RUNG wire#powerrail
      I_Contact( "AI_PLC1_Step_Bon1_Dosing" )
      { S7_GenerateENO := "TRUE" } Move(in := 0.0, out1 => "AI_CV3201_Nuoc_Bon1")
   END_RUNG
   // the same network as SCL:
   IF NOT "AI_PLC1_Step_Bon1_Dosing" THEN "AI_CV3201_Nuoc_Bon1" := 0.0; END_IF;
END_REGION

REGION Network 165: Reset CV nước Bồn 1 khi Stop hoặc Lỗi tổng PLC1
   RUNG wire#powerrail
      Contact( "AI_PLC1_Stop_Active" )
      wire#w1
      { S7_GenerateENO := "TRUE" } Move(in := 0.0, out1 => "AI_CV3201_Nuoc_Bon1")
   END_RUNG
   RUNG wire#powerrail
      Contact( "AI_PLC1_Loi_Tong" )
   END_RUNG wire#w1
   // the same network as SCL:
   IF "AI_PLC1_Stop_Active" OR "AI_PLC1_Loi_Tong" THEN "AI_CV3201_Nuoc_Bon1" := 0.0; END_IF;
END_REGION

REGION Network 166: Clamp CV nước Bồn 1 trong dải 0.0-100.0 (Dưới)
   RUNG wire#powerrail
      { S7_Templates := "SrcType := Real" } LT_Contact(in1 := "AI_CV3201_Nuoc_Bon1", in2 := 0.0)
      { S7_GenerateENO := "TRUE" } Move(in := 0.0, out1 => "AI_CV3201_Nuoc_Bon1")
   END_RUNG
   // the same network as SCL:
   IF "AI_CV3201_Nuoc_Bon1" < 0.0 THEN "AI_CV3201_Nuoc_Bon1" := 0.0; END_IF;
END_REGION

REGION Network 167: Clamp CV nước Bồn 1 trong dải 0.0-100.0 (Trên)
   RUNG wire#powerrail
      { S7_Templates := "SrcType := Real" } GT_Contact(in1 := "AI_CV3201_Nuoc_Bon1", in2 := 100.0)
      { S7_GenerateENO := "TRUE" } Move(in := 100.0, out1 => "AI_CV3201_Nuoc_Bon1")
   END_RUNG
   // the same network as SCL:
   IF "AI_CV3201_Nuoc_Bon1" > 100.0 THEN "AI_CV3201_Nuoc_Bon1" := 100.0; END_IF;
END_REGION

REGION Network 168: Reset tốc độ cánh khuấy Bồn 1 khi không khuấy
   RUNG wire#powerrail
      I_Contact( "AI_PLC1_Step_Bon1_Khuay" )
      { S7_GenerateENO := "TRUE" } Move(in := 0.0, out1 => "AI_AGTR3260_Toc_Do_AO")
   END_RUNG
   // the same network as SCL:
   IF NOT "AI_PLC1_Step_Bon1_Khuay" THEN "AI_AGTR3260_Toc_Do_AO" := 0.0; END_IF;
END_REGION

REGION Network 169: Reset tốc độ cánh khuấy Bồn 1 khi Stop hoặc Lỗi tổng PLC1
   RUNG wire#powerrail
      Contact( "AI_PLC1_Stop_Active" )
      wire#w1
      { S7_GenerateENO := "TRUE" } Move(in := 0.0, out1 => "AI_AGTR3260_Toc_Do_AO")
   END_RUNG
   RUNG wire#powerrail
      Contact( "AI_PLC1_Loi_Tong" )
   END_RUNG wire#w1
   // the same network as SCL:
   IF "AI_PLC1_Stop_Active" OR "AI_PLC1_Loi_Tong" THEN "AI_AGTR3260_Toc_Do_AO" := 0.0; END_IF;
END_REGION

REGION Network 170: Clamp tốc độ cánh khuấy Bồn 1 trong dải 0.0-100.0 (Dưới)
   RUNG wire#powerrail
      { S7_Templates := "SrcType := Real" } LT_Contact(in1 := "AI_AGTR3260_Toc_Do_AO", in2 := 0.0)
      { S7_GenerateENO := "TRUE" } Move(in := 0.0, out1 => "AI_AGTR3260_Toc_Do_AO")
   END_RUNG
   // the same network as SCL:
   IF "AI_AGTR3260_Toc_Do_AO" < 0.0 THEN "AI_AGTR3260_Toc_Do_AO" := 0.0; END_IF;
END_REGION

REGION Network 171: Clamp tốc độ cánh khuấy Bồn 1 trong dải 0.0-100.0 (Trên)
   RUNG wire#powerrail
      { S7_Templates := "SrcType := Real" } GT_Contact(in1 := "AI_AGTR3260_Toc_Do_AO", in2 := 100.0)
      { S7_GenerateENO := "TRUE" } Move(in := 100.0, out1 => "AI_AGTR3260_Toc_Do_AO")
   END_RUNG
   // the same network as SCL:
   IF "AI_AGTR3260_Toc_Do_AO" > 100.0 THEN "AI_AGTR3260_Toc_Do_AO" := 100.0; END_IF;
END_REGION

REGION Network 172: Reset CV hơi Bồn 2 khi không chạy PID
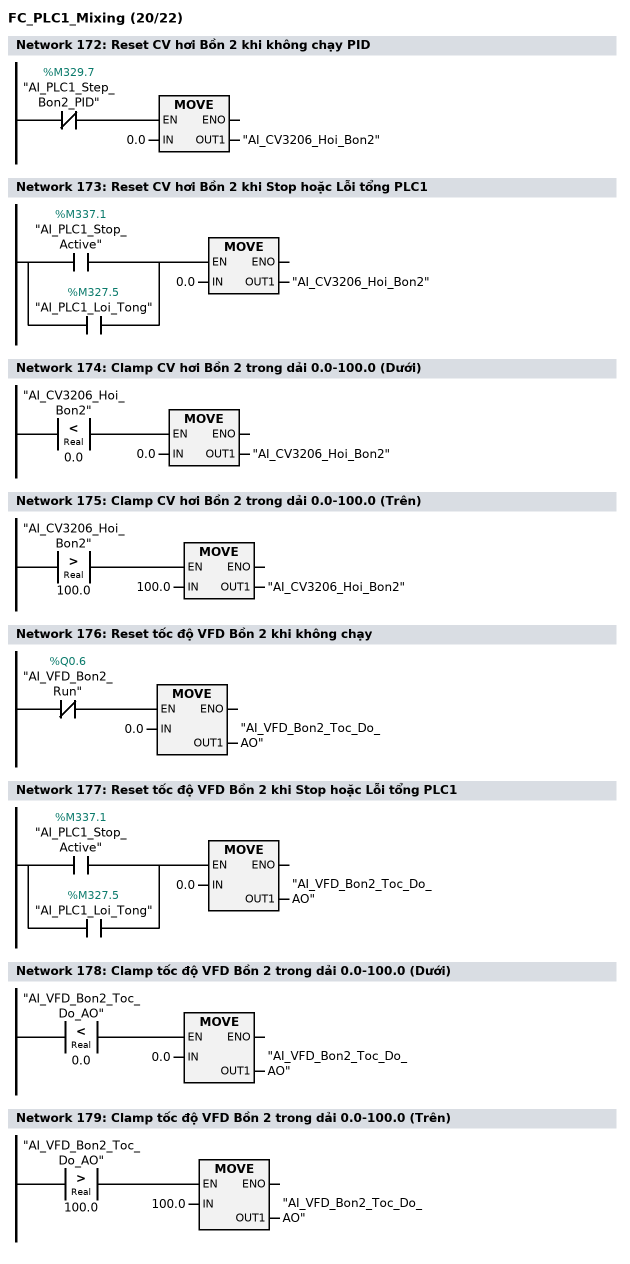
   RUNG wire#powerrail
      I_Contact( "AI_PLC1_Step_Bon2_PID" )
      { S7_GenerateENO := "TRUE" } Move(in := 0.0, out1 => "AI_CV3206_Hoi_Bon2")
   END_RUNG
   // the same network as SCL:
   IF NOT "AI_PLC1_Step_Bon2_PID" THEN "AI_CV3206_Hoi_Bon2" := 0.0; END_IF;
END_REGION

REGION Network 173: Reset CV hơi Bồn 2 khi Stop hoặc Lỗi tổng PLC1
   RUNG wire#powerrail
      Contact( "AI_PLC1_Stop_Active" )
      wire#w1
      { S7_GenerateENO := "TRUE" } Move(in := 0.0, out1 => "AI_CV3206_Hoi_Bon2")
   END_RUNG
   RUNG wire#powerrail
      Contact( "AI_PLC1_Loi_Tong" )
   END_RUNG wire#w1
   // the same network as SCL:
   IF "AI_PLC1_Stop_Active" OR "AI_PLC1_Loi_Tong" THEN "AI_CV3206_Hoi_Bon2" := 0.0; END_IF;
END_REGION

REGION Network 174: Clamp CV hơi Bồn 2 trong dải 0.0-100.0 (Dưới)
   RUNG wire#powerrail
      { S7_Templates := "SrcType := Real" } LT_Contact(in1 := "AI_CV3206_Hoi_Bon2", in2 := 0.0)
      { S7_GenerateENO := "TRUE" } Move(in := 0.0, out1 => "AI_CV3206_Hoi_Bon2")
   END_RUNG
   // the same network as SCL:
   IF "AI_CV3206_Hoi_Bon2" < 0.0 THEN "AI_CV3206_Hoi_Bon2" := 0.0; END_IF;
END_REGION

REGION Network 175: Clamp CV hơi Bồn 2 trong dải 0.0-100.0 (Trên)
   RUNG wire#powerrail
      { S7_Templates := "SrcType := Real" } GT_Contact(in1 := "AI_CV3206_Hoi_Bon2", in2 := 100.0)
      { S7_GenerateENO := "TRUE" } Move(in := 100.0, out1 => "AI_CV3206_Hoi_Bon2")
   END_RUNG
   // the same network as SCL:
   IF "AI_CV3206_Hoi_Bon2" > 100.0 THEN "AI_CV3206_Hoi_Bon2" := 100.0; END_IF;
END_REGION

REGION Network 176: Reset tốc độ VFD Bồn 2 khi không chạy
   RUNG wire#powerrail
      I_Contact( "AI_VFD_Bon2_Run" )
      { S7_GenerateENO := "TRUE" } Move(in := 0.0, out1 => "AI_VFD_Bon2_Toc_Do_AO")
   END_RUNG
   // the same network as SCL:
   IF NOT "AI_VFD_Bon2_Run" THEN "AI_VFD_Bon2_Toc_Do_AO" := 0.0; END_IF;
END_REGION

REGION Network 177: Reset tốc độ VFD Bồn 2 khi Stop hoặc Lỗi tổng PLC1
   RUNG wire#powerrail
      Contact( "AI_PLC1_Stop_Active" )
      wire#w1
      { S7_GenerateENO := "TRUE" } Move(in := 0.0, out1 => "AI_VFD_Bon2_Toc_Do_AO")
   END_RUNG
   RUNG wire#powerrail
      Contact( "AI_PLC1_Loi_Tong" )
   END_RUNG wire#w1
   // the same network as SCL:
   IF "AI_PLC1_Stop_Active" OR "AI_PLC1_Loi_Tong" THEN "AI_VFD_Bon2_Toc_Do_AO" := 0.0; END_IF;
END_REGION

REGION Network 178: Clamp tốc độ VFD Bồn 2 trong dải 0.0-100.0 (Dưới)
   RUNG wire#powerrail
      { S7_Templates := "SrcType := Real" } LT_Contact(in1 := "AI_VFD_Bon2_Toc_Do_AO", in2 := 0.0)
      { S7_GenerateENO := "TRUE" } Move(in := 0.0, out1 => "AI_VFD_Bon2_Toc_Do_AO")
   END_RUNG
   // the same network as SCL:
   IF "AI_VFD_Bon2_Toc_Do_AO" < 0.0 THEN "AI_VFD_Bon2_Toc_Do_AO" := 0.0; END_IF;
END_REGION

REGION Network 179: Clamp tốc độ VFD Bồn 2 trong dải 0.0-100.0 (Trên)
   RUNG wire#powerrail
      { S7_Templates := "SrcType := Real" } GT_Contact(in1 := "AI_VFD_Bon2_Toc_Do_AO", in2 := 100.0)
      { S7_GenerateENO := "TRUE" } Move(in := 100.0, out1 => "AI_VFD_Bon2_Toc_Do_AO")
   END_RUNG
   // the same network as SCL:
   IF "AI_VFD_Bon2_Toc_Do_AO" > 100.0 THEN "AI_VFD_Bon2_Toc_Do_AO" := 100.0; END_IF;
END_REGION

REGION Network 180: VFD Bon 2 Freq Scale: Speed SP x 5.0
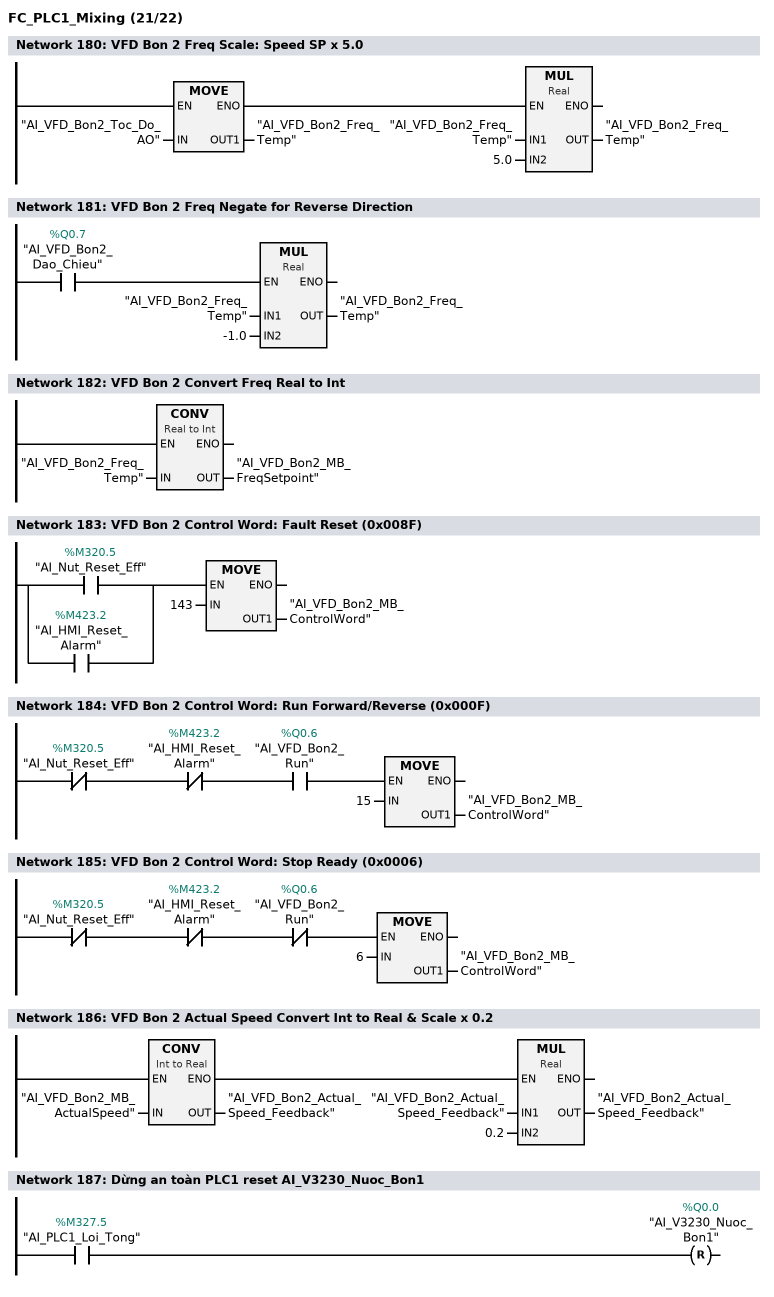
   RUNG wire#powerrail
      { S7_GenerateENO := "TRUE" } Move(in := "AI_VFD_Bon2_Toc_Do_AO", out1 => "AI_VFD_Bon2_Freq_Temp")
      { S7_Templates := "SrcType := Real"; S7_GenerateENO := "TRUE" } Mul(in1 := "AI_VFD_Bon2_Freq_Temp", in2 := 5.0, out => "AI_VFD_Bon2_Freq_Temp")
   END_RUNG
   // the same network as SCL:
   // ENO of a box is taken as its EN; it also drops when the box reports an error
   "AI_VFD_Bon2_Freq_Temp" := "AI_VFD_Bon2_Toc_Do_AO";
   "AI_VFD_Bon2_Freq_Temp" := "AI_VFD_Bon2_Freq_Temp" * 5.0;
END_REGION

REGION Network 181: VFD Bon 2 Freq Negate for Reverse Direction
   RUNG wire#powerrail
      Contact( "AI_VFD_Bon2_Dao_Chieu" )
      { S7_Templates := "SrcType := Real"; S7_GenerateENO := "TRUE" } Mul(in1 := "AI_VFD_Bon2_Freq_Temp", in2 := -1.0, out => "AI_VFD_Bon2_Freq_Temp")
   END_RUNG
   // the same network as SCL:
   IF "AI_VFD_Bon2_Dao_Chieu" THEN "AI_VFD_Bon2_Freq_Temp" := "AI_VFD_Bon2_Freq_Temp" * (-1.0); END_IF;
END_REGION

REGION Network 182: VFD Bon 2 Convert Freq Real to Int
   RUNG wire#powerrail
      { S7_Templates := "[SrcType := Real, DestType := Int]"; S7_GenerateENO := "TRUE" } Convert(in := "AI_VFD_Bon2_Freq_Temp", out => "AI_VFD_Bon2_MB_FreqSetpoint")
   END_RUNG
   // the same network as SCL:
   "AI_VFD_Bon2_MB_FreqSetpoint" := REAL_TO_INT("AI_VFD_Bon2_Freq_Temp");
END_REGION

REGION Network 183: VFD Bon 2 Control Word: Fault Reset (0x008F)
   RUNG wire#powerrail
      Contact( "AI_Nut_Reset_Eff" )
      wire#w1
      { S7_GenerateENO := "TRUE" } Move(in := 143, out1 => "AI_VFD_Bon2_MB_ControlWord")
   END_RUNG
   RUNG wire#powerrail
      Contact( "AI_HMI_Reset_Alarm" )
   END_RUNG wire#w1
   // the same network as SCL:
   IF "AI_Nut_Reset_Eff" OR "AI_HMI_Reset_Alarm" THEN "AI_VFD_Bon2_MB_ControlWord" := 143; END_IF;
END_REGION

REGION Network 184: VFD Bon 2 Control Word: Run Forward/Reverse (0x000F)
   RUNG wire#powerrail
      I_Contact( "AI_Nut_Reset_Eff" )
      I_Contact( "AI_HMI_Reset_Alarm" )
      Contact( "AI_VFD_Bon2_Run" )
      { S7_GenerateENO := "TRUE" } Move(in := 15, out1 => "AI_VFD_Bon2_MB_ControlWord")
   END_RUNG
   // the same network as SCL:
   IF NOT "AI_Nut_Reset_Eff" AND NOT "AI_HMI_Reset_Alarm" AND "AI_VFD_Bon2_Run" THEN
       "AI_VFD_Bon2_MB_ControlWord" := 15;
   END_IF;
END_REGION

REGION Network 185: VFD Bon 2 Control Word: Stop Ready (0x0006)
   RUNG wire#powerrail
      I_Contact( "AI_Nut_Reset_Eff" )
      I_Contact( "AI_HMI_Reset_Alarm" )
      I_Contact( "AI_VFD_Bon2_Run" )
      { S7_GenerateENO := "TRUE" } Move(in := 6, out1 => "AI_VFD_Bon2_MB_ControlWord")
   END_RUNG
   // the same network as SCL:
   IF NOT "AI_Nut_Reset_Eff" AND NOT "AI_HMI_Reset_Alarm" AND NOT "AI_VFD_Bon2_Run" THEN
       "AI_VFD_Bon2_MB_ControlWord" := 6;
   END_IF;
END_REGION

REGION Network 186: VFD Bon 2 Actual Speed Convert Int to Real & Scale x 0.2
   RUNG wire#powerrail
      { S7_Templates := "[SrcType := Int, DestType := Real]"; S7_GenerateENO := "TRUE" } Convert(in := "AI_VFD_Bon2_MB_ActualSpeed", out => "AI_VFD_Bon2_Actual_Speed_Feedback")
      { S7_Templates := "SrcType := Real"; S7_GenerateENO := "TRUE" } Mul(in1 := "AI_VFD_Bon2_Actual_Speed_Feedback", in2 := 0.2, out => "AI_VFD_Bon2_Actual_Speed_Feedback")
   END_RUNG
   // the same network as SCL:
   // ENO of a box is taken as its EN; it also drops when the box reports an error
   "AI_VFD_Bon2_Actual_Speed_Feedback" := INT_TO_REAL("AI_VFD_Bon2_MB_ActualSpeed");
   "AI_VFD_Bon2_Actual_Speed_Feedback" := "AI_VFD_Bon2_Actual_Speed_Feedback" * 0.2;
END_REGION

REGION Network 187: Dừng an toàn PLC1 reset AI_V3230_Nuoc_Bon1
   RUNG wire#powerrail
      Contact( "AI_PLC1_Loi_Tong" )
      R_Coil( "AI_V3230_Nuoc_Bon1" )
   END_RUNG
   // the same network as SCL:
   IF "AI_PLC1_Loi_Tong" THEN "AI_V3230_Nuoc_Bon1" := FALSE; END_IF;
END_REGION

REGION Network 188: Dừng an toàn PLC1 reset AI_V3232_Xa_Bon1
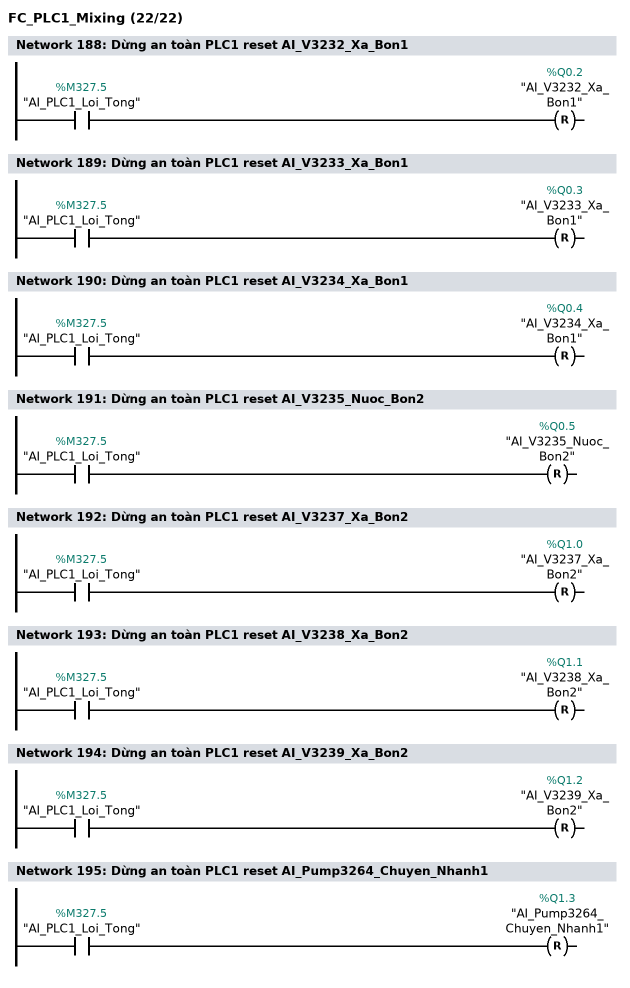
   RUNG wire#powerrail
      Contact( "AI_PLC1_Loi_Tong" )
      R_Coil( "AI_V3232_Xa_Bon1" )
   END_RUNG
   // the same network as SCL:
   IF "AI_PLC1_Loi_Tong" THEN "AI_V3232_Xa_Bon1" := FALSE; END_IF;
END_REGION

REGION Network 189: Dừng an toàn PLC1 reset AI_V3233_Xa_Bon1
   RUNG wire#powerrail
      Contact( "AI_PLC1_Loi_Tong" )
      R_Coil( "AI_V3233_Xa_Bon1" )
   END_RUNG
   // the same network as SCL:
   IF "AI_PLC1_Loi_Tong" THEN "AI_V3233_Xa_Bon1" := FALSE; END_IF;
END_REGION

REGION Network 190: Dừng an toàn PLC1 reset AI_V3234_Xa_Bon1
   RUNG wire#powerrail
      Contact( "AI_PLC1_Loi_Tong" )
      R_Coil( "AI_V3234_Xa_Bon1" )
   END_RUNG
   // the same network as SCL:
   IF "AI_PLC1_Loi_Tong" THEN "AI_V3234_Xa_Bon1" := FALSE; END_IF;
END_REGION

REGION Network 191: Dừng an toàn PLC1 reset AI_V3235_Nuoc_Bon2
   RUNG wire#powerrail
      Contact( "AI_PLC1_Loi_Tong" )
      R_Coil( "AI_V3235_Nuoc_Bon2" )
   END_RUNG
   // the same network as SCL:
   IF "AI_PLC1_Loi_Tong" THEN "AI_V3235_Nuoc_Bon2" := FALSE; END_IF;
END_REGION

REGION Network 192: Dừng an toàn PLC1 reset AI_V3237_Xa_Bon2
   RUNG wire#powerrail
      Contact( "AI_PLC1_Loi_Tong" )
      R_Coil( "AI_V3237_Xa_Bon2" )
   END_RUNG
   // the same network as SCL:
   IF "AI_PLC1_Loi_Tong" THEN "AI_V3237_Xa_Bon2" := FALSE; END_IF;
END_REGION

REGION Network 193: Dừng an toàn PLC1 reset AI_V3238_Xa_Bon2
   RUNG wire#powerrail
      Contact( "AI_PLC1_Loi_Tong" )
      R_Coil( "AI_V3238_Xa_Bon2" )
   END_RUNG
   // the same network as SCL:
   IF "AI_PLC1_Loi_Tong" THEN "AI_V3238_Xa_Bon2" := FALSE; END_IF;
END_REGION

REGION Network 194: Dừng an toàn PLC1 reset AI_V3239_Xa_Bon2
   RUNG wire#powerrail
      Contact( "AI_PLC1_Loi_Tong" )
      R_Coil( "AI_V3239_Xa_Bon2" )
   END_RUNG
   // the same network as SCL:
   IF "AI_PLC1_Loi_Tong" THEN "AI_V3239_Xa_Bon2" := FALSE; END_IF;
END_REGION

REGION Network 195: Dừng an toàn PLC1 reset AI_Pump3264_Chuyen_Nhanh1
   RUNG wire#powerrail
      Contact( "AI_PLC1_Loi_Tong" )
      R_Coil( "AI_Pump3264_Chuyen_Nhanh1" )
   END_RUNG
   // the same network as SCL:
   IF "AI_PLC1_Loi_Tong" THEN "AI_Pump3264_Chuyen_Nhanh1" := FALSE; END_IF;
END_REGION
END_FUNCTION

FUNCTION "FC_Bon_Chua_Loc" : Void   // FC30, LAD
{ S7_Optimized_Access := 'TRUE' }
VERSION : 0.1
// stored: AutoNumber true, IsIECCheckEnabled false, SetENOAutomatically false, UDAEnableTagReadback false
BEGIN

REGION Network 1: Gated HMI AI_LSH3310_Pheu_Cao qua Sim Mode
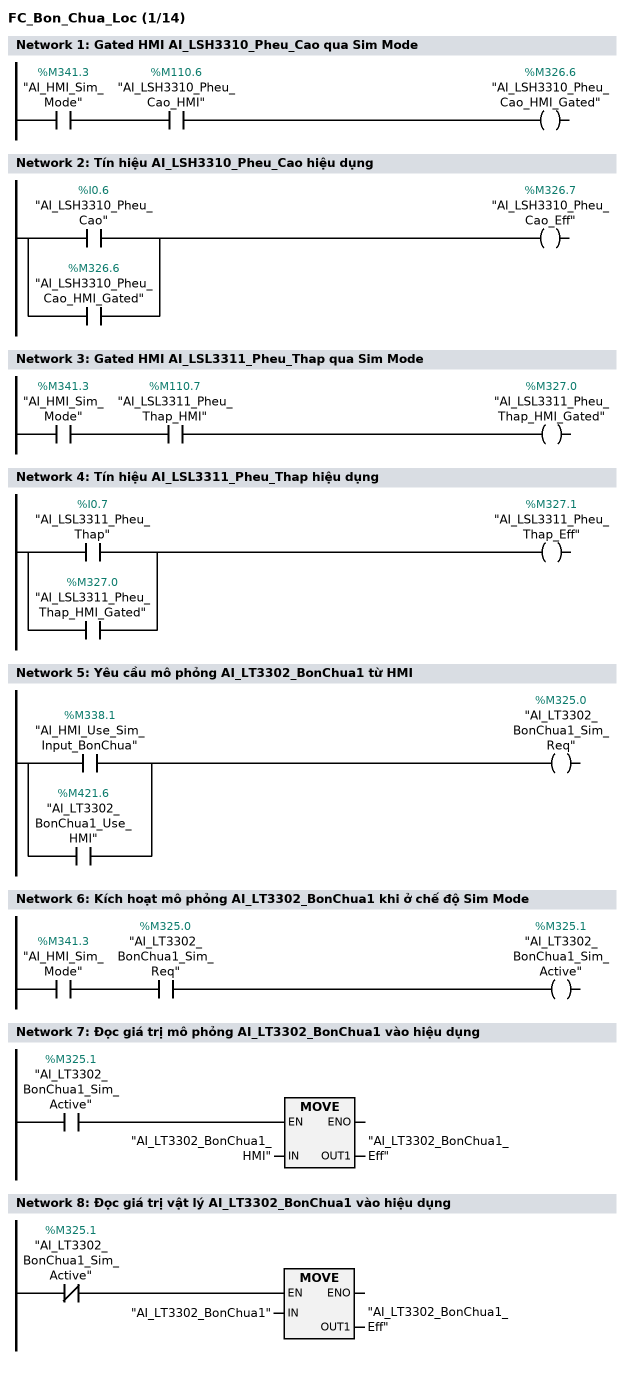
   RUNG wire#powerrail
      Contact( "AI_HMI_Sim_Mode" )
      Contact( "AI_LSH3310_Pheu_Cao_HMI" )
      Coil( "AI_LSH3310_Pheu_Cao_HMI_Gated" )
   END_RUNG
   // the same network as SCL:
   "AI_LSH3310_Pheu_Cao_HMI_Gated" := "AI_HMI_Sim_Mode" AND "AI_LSH3310_Pheu_Cao_HMI";
END_REGION

REGION Network 2: Tín hiệu AI_LSH3310_Pheu_Cao hiệu dụng
   RUNG wire#powerrail
      Contact( "AI_LSH3310_Pheu_Cao" )
      wire#w1
      Coil( "AI_LSH3310_Pheu_Cao_Eff" )
   END_RUNG
   RUNG wire#powerrail
      Contact( "AI_LSH3310_Pheu_Cao_HMI_Gated" )
   END_RUNG wire#w1
   // the same network as SCL:
   "AI_LSH3310_Pheu_Cao_Eff" := "AI_LSH3310_Pheu_Cao" OR "AI_LSH3310_Pheu_Cao_HMI_Gated";
END_REGION

REGION Network 3: Gated HMI AI_LSL3311_Pheu_Thap qua Sim Mode
   RUNG wire#powerrail
      Contact( "AI_HMI_Sim_Mode" )
      Contact( "AI_LSL3311_Pheu_Thap_HMI" )
      Coil( "AI_LSL3311_Pheu_Thap_HMI_Gated" )
   END_RUNG
   // the same network as SCL:
   "AI_LSL3311_Pheu_Thap_HMI_Gated" := "AI_HMI_Sim_Mode" AND "AI_LSL3311_Pheu_Thap_HMI";
END_REGION

REGION Network 4: Tín hiệu AI_LSL3311_Pheu_Thap hiệu dụng
   RUNG wire#powerrail
      Contact( "AI_LSL3311_Pheu_Thap" )
      wire#w1
      Coil( "AI_LSL3311_Pheu_Thap_Eff" )
   END_RUNG
   RUNG wire#powerrail
      Contact( "AI_LSL3311_Pheu_Thap_HMI_Gated" )
   END_RUNG wire#w1
   // the same network as SCL:
   "AI_LSL3311_Pheu_Thap_Eff" := "AI_LSL3311_Pheu_Thap" OR "AI_LSL3311_Pheu_Thap_HMI_Gated";
END_REGION

REGION Network 5: Yêu cầu mô phỏng AI_LT3302_BonChua1 từ HMI
   RUNG wire#powerrail
      Contact( "AI_HMI_Use_Sim_Input_BonChua" )
      wire#w1
      Coil( "AI_LT3302_BonChua1_Sim_Req" )
   END_RUNG
   RUNG wire#powerrail
      Contact( "AI_LT3302_BonChua1_Use_HMI" )
   END_RUNG wire#w1
   // the same network as SCL:
   "AI_LT3302_BonChua1_Sim_Req" := "AI_HMI_Use_Sim_Input_BonChua" OR "AI_LT3302_BonChua1_Use_HMI";
END_REGION

REGION Network 6: Kích hoạt mô phỏng AI_LT3302_BonChua1 khi ở chế độ Sim Mode
   RUNG wire#powerrail
      Contact( "AI_HMI_Sim_Mode" )
      Contact( "AI_LT3302_BonChua1_Sim_Req" )
      Coil( "AI_LT3302_BonChua1_Sim_Active" )
   END_RUNG
   // the same network as SCL:
   "AI_LT3302_BonChua1_Sim_Active" := "AI_HMI_Sim_Mode" AND "AI_LT3302_BonChua1_Sim_Req";
END_REGION

REGION Network 7: Đọc giá trị mô phỏng AI_LT3302_BonChua1 vào hiệu dụng
   RUNG wire#powerrail
      Contact( "AI_LT3302_BonChua1_Sim_Active" )
      { S7_GenerateENO := "TRUE" } Move(in := "AI_LT3302_BonChua1_HMI", out1 => "AI_LT3302_BonChua1_Eff")
   END_RUNG
   // the same network as SCL:
   IF "AI_LT3302_BonChua1_Sim_Active" THEN "AI_LT3302_BonChua1_Eff" := "AI_LT3302_BonChua1_HMI"; END_IF;
END_REGION

REGION Network 8: Đọc giá trị vật lý AI_LT3302_BonChua1 vào hiệu dụng
   RUNG wire#powerrail
      I_Contact( "AI_LT3302_BonChua1_Sim_Active" )
      { S7_GenerateENO := "TRUE" } Move(in := "AI_LT3302_BonChua1", out1 => "AI_LT3302_BonChua1_Eff")
   END_RUNG
   // the same network as SCL:
   IF NOT "AI_LT3302_BonChua1_Sim_Active" THEN "AI_LT3302_BonChua1_Eff" := "AI_LT3302_BonChua1"; END_IF;
END_REGION

REGION Network 9: Yêu cầu mô phỏng AI_TT3301_BonChua1 từ HMI
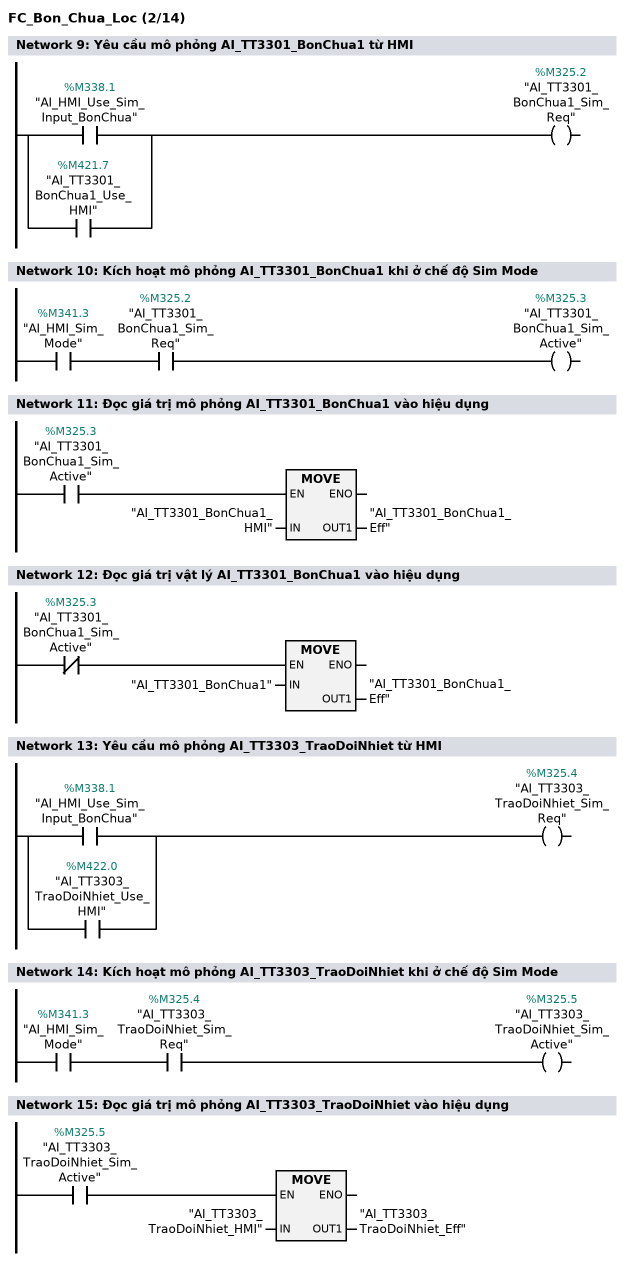
   RUNG wire#powerrail
      Contact( "AI_HMI_Use_Sim_Input_BonChua" )
      wire#w1
      Coil( "AI_TT3301_BonChua1_Sim_Req" )
   END_RUNG
   RUNG wire#powerrail
      Contact( "AI_TT3301_BonChua1_Use_HMI" )
   END_RUNG wire#w1
   // the same network as SCL:
   "AI_TT3301_BonChua1_Sim_Req" := "AI_HMI_Use_Sim_Input_BonChua" OR "AI_TT3301_BonChua1_Use_HMI";
END_REGION

REGION Network 10: Kích hoạt mô phỏng AI_TT3301_BonChua1 khi ở chế độ Sim Mode
   RUNG wire#powerrail
      Contact( "AI_HMI_Sim_Mode" )
      Contact( "AI_TT3301_BonChua1_Sim_Req" )
      Coil( "AI_TT3301_BonChua1_Sim_Active" )
   END_RUNG
   // the same network as SCL:
   "AI_TT3301_BonChua1_Sim_Active" := "AI_HMI_Sim_Mode" AND "AI_TT3301_BonChua1_Sim_Req";
END_REGION

REGION Network 11: Đọc giá trị mô phỏng AI_TT3301_BonChua1 vào hiệu dụng
   RUNG wire#powerrail
      Contact( "AI_TT3301_BonChua1_Sim_Active" )
      { S7_GenerateENO := "TRUE" } Move(in := "AI_TT3301_BonChua1_HMI", out1 => "AI_TT3301_BonChua1_Eff")
   END_RUNG
   // the same network as SCL:
   IF "AI_TT3301_BonChua1_Sim_Active" THEN "AI_TT3301_BonChua1_Eff" := "AI_TT3301_BonChua1_HMI"; END_IF;
END_REGION

REGION Network 12: Đọc giá trị vật lý AI_TT3301_BonChua1 vào hiệu dụng
   RUNG wire#powerrail
      I_Contact( "AI_TT3301_BonChua1_Sim_Active" )
      { S7_GenerateENO := "TRUE" } Move(in := "AI_TT3301_BonChua1", out1 => "AI_TT3301_BonChua1_Eff")
   END_RUNG
   // the same network as SCL:
   IF NOT "AI_TT3301_BonChua1_Sim_Active" THEN "AI_TT3301_BonChua1_Eff" := "AI_TT3301_BonChua1"; END_IF;
END_REGION

REGION Network 13: Yêu cầu mô phỏng AI_TT3303_TraoDoiNhiet từ HMI
   RUNG wire#powerrail
      Contact( "AI_HMI_Use_Sim_Input_BonChua" )
      wire#w1
      Coil( "AI_TT3303_TraoDoiNhiet_Sim_Req" )
   END_RUNG
   RUNG wire#powerrail
      Contact( "AI_TT3303_TraoDoiNhiet_Use_HMI" )
   END_RUNG wire#w1
   // the same network as SCL:
   "AI_TT3303_TraoDoiNhiet_Sim_Req" := "AI_HMI_Use_Sim_Input_BonChua" OR "AI_TT3303_TraoDoiNhiet_Use_HMI";
END_REGION

REGION Network 14: Kích hoạt mô phỏng AI_TT3303_TraoDoiNhiet khi ở chế độ Sim Mode
   RUNG wire#powerrail
      Contact( "AI_HMI_Sim_Mode" )
      Contact( "AI_TT3303_TraoDoiNhiet_Sim_Req" )
      Coil( "AI_TT3303_TraoDoiNhiet_Sim_Active" )
   END_RUNG
   // the same network as SCL:
   "AI_TT3303_TraoDoiNhiet_Sim_Active" := "AI_HMI_Sim_Mode" AND "AI_TT3303_TraoDoiNhiet_Sim_Req";
END_REGION

REGION Network 15: Đọc giá trị mô phỏng AI_TT3303_TraoDoiNhiet vào hiệu dụng
   RUNG wire#powerrail
      Contact( "AI_TT3303_TraoDoiNhiet_Sim_Active" )
      { S7_GenerateENO := "TRUE" } Move(in := "AI_TT3303_TraoDoiNhiet_HMI", out1 => "AI_TT3303_TraoDoiNhiet_Eff")
   END_RUNG
   // the same network as SCL:
   IF "AI_TT3303_TraoDoiNhiet_Sim_Active" THEN
       "AI_TT3303_TraoDoiNhiet_Eff" := "AI_TT3303_TraoDoiNhiet_HMI";
   END_IF;
END_REGION

REGION Network 16: Đọc giá trị vật lý AI_TT3303_TraoDoiNhiet vào hiệu dụng
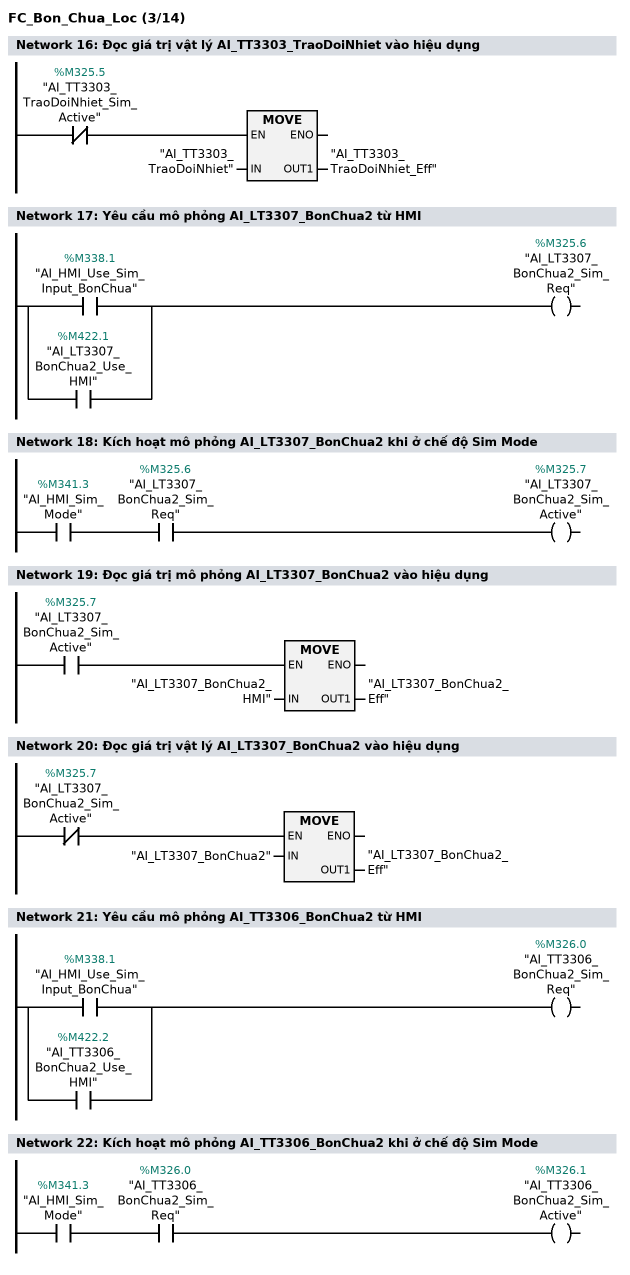
   RUNG wire#powerrail
      I_Contact( "AI_TT3303_TraoDoiNhiet_Sim_Active" )
      { S7_GenerateENO := "TRUE" } Move(in := "AI_TT3303_TraoDoiNhiet", out1 => "AI_TT3303_TraoDoiNhiet_Eff")
   END_RUNG
   // the same network as SCL:
   IF NOT "AI_TT3303_TraoDoiNhiet_Sim_Active" THEN
       "AI_TT3303_TraoDoiNhiet_Eff" := "AI_TT3303_TraoDoiNhiet";
   END_IF;
END_REGION

REGION Network 17: Yêu cầu mô phỏng AI_LT3307_BonChua2 từ HMI
   RUNG wire#powerrail
      Contact( "AI_HMI_Use_Sim_Input_BonChua" )
      wire#w1
      Coil( "AI_LT3307_BonChua2_Sim_Req" )
   END_RUNG
   RUNG wire#powerrail
      Contact( "AI_LT3307_BonChua2_Use_HMI" )
   END_RUNG wire#w1
   // the same network as SCL:
   "AI_LT3307_BonChua2_Sim_Req" := "AI_HMI_Use_Sim_Input_BonChua" OR "AI_LT3307_BonChua2_Use_HMI";
END_REGION

REGION Network 18: Kích hoạt mô phỏng AI_LT3307_BonChua2 khi ở chế độ Sim Mode
   RUNG wire#powerrail
      Contact( "AI_HMI_Sim_Mode" )
      Contact( "AI_LT3307_BonChua2_Sim_Req" )
      Coil( "AI_LT3307_BonChua2_Sim_Active" )
   END_RUNG
   // the same network as SCL:
   "AI_LT3307_BonChua2_Sim_Active" := "AI_HMI_Sim_Mode" AND "AI_LT3307_BonChua2_Sim_Req";
END_REGION

REGION Network 19: Đọc giá trị mô phỏng AI_LT3307_BonChua2 vào hiệu dụng
   RUNG wire#powerrail
      Contact( "AI_LT3307_BonChua2_Sim_Active" )
      { S7_GenerateENO := "TRUE" } Move(in := "AI_LT3307_BonChua2_HMI", out1 => "AI_LT3307_BonChua2_Eff")
   END_RUNG
   // the same network as SCL:
   IF "AI_LT3307_BonChua2_Sim_Active" THEN "AI_LT3307_BonChua2_Eff" := "AI_LT3307_BonChua2_HMI"; END_IF;
END_REGION

REGION Network 20: Đọc giá trị vật lý AI_LT3307_BonChua2 vào hiệu dụng
   RUNG wire#powerrail
      I_Contact( "AI_LT3307_BonChua2_Sim_Active" )
      { S7_GenerateENO := "TRUE" } Move(in := "AI_LT3307_BonChua2", out1 => "AI_LT3307_BonChua2_Eff")
   END_RUNG
   // the same network as SCL:
   IF NOT "AI_LT3307_BonChua2_Sim_Active" THEN "AI_LT3307_BonChua2_Eff" := "AI_LT3307_BonChua2"; END_IF;
END_REGION

REGION Network 21: Yêu cầu mô phỏng AI_TT3306_BonChua2 từ HMI
   RUNG wire#powerrail
      Contact( "AI_HMI_Use_Sim_Input_BonChua" )
      wire#w1
      Coil( "AI_TT3306_BonChua2_Sim_Req" )
   END_RUNG
   RUNG wire#powerrail
      Contact( "AI_TT3306_BonChua2_Use_HMI" )
   END_RUNG wire#w1
   // the same network as SCL:
   "AI_TT3306_BonChua2_Sim_Req" := "AI_HMI_Use_Sim_Input_BonChua" OR "AI_TT3306_BonChua2_Use_HMI";
END_REGION

REGION Network 22: Kích hoạt mô phỏng AI_TT3306_BonChua2 khi ở chế độ Sim Mode
   RUNG wire#powerrail
      Contact( "AI_HMI_Sim_Mode" )
      Contact( "AI_TT3306_BonChua2_Sim_Req" )
      Coil( "AI_TT3306_BonChua2_Sim_Active" )
   END_RUNG
   // the same network as SCL:
   "AI_TT3306_BonChua2_Sim_Active" := "AI_HMI_Sim_Mode" AND "AI_TT3306_BonChua2_Sim_Req";
END_REGION

REGION Network 23: Đọc giá trị mô phỏng AI_TT3306_BonChua2 vào hiệu dụng
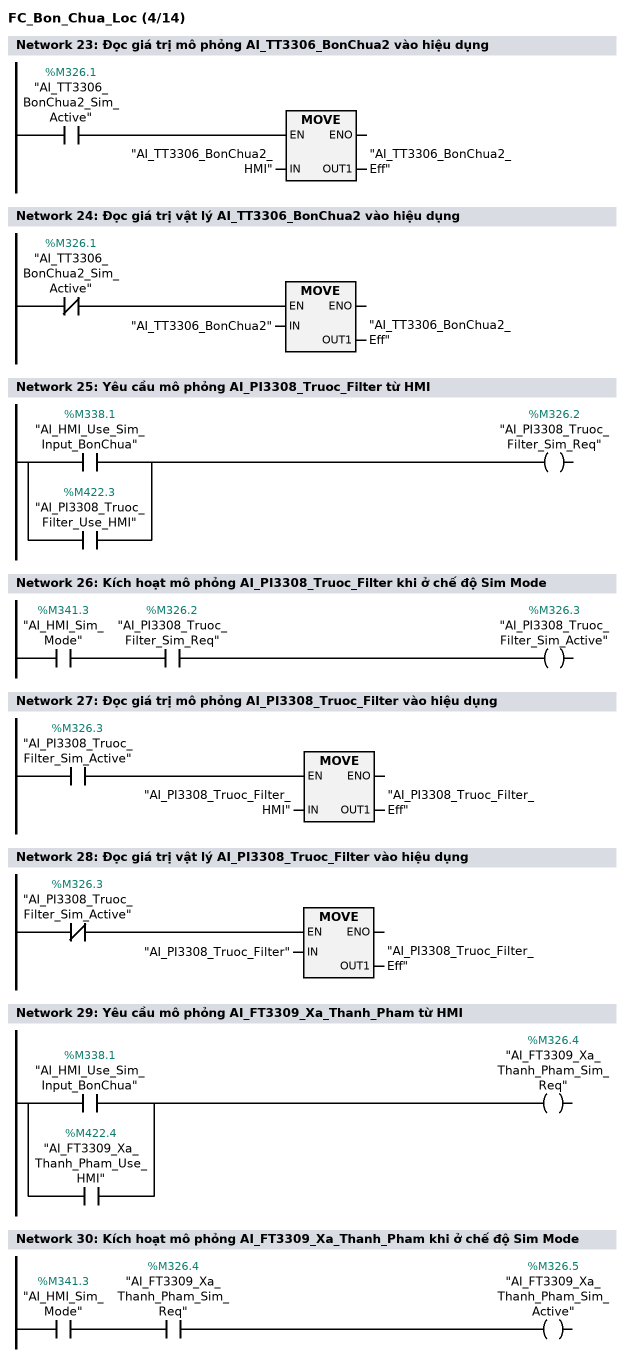
   RUNG wire#powerrail
      Contact( "AI_TT3306_BonChua2_Sim_Active" )
      { S7_GenerateENO := "TRUE" } Move(in := "AI_TT3306_BonChua2_HMI", out1 => "AI_TT3306_BonChua2_Eff")
   END_RUNG
   // the same network as SCL:
   IF "AI_TT3306_BonChua2_Sim_Active" THEN "AI_TT3306_BonChua2_Eff" := "AI_TT3306_BonChua2_HMI"; END_IF;
END_REGION

REGION Network 24: Đọc giá trị vật lý AI_TT3306_BonChua2 vào hiệu dụng
   RUNG wire#powerrail
      I_Contact( "AI_TT3306_BonChua2_Sim_Active" )
      { S7_GenerateENO := "TRUE" } Move(in := "AI_TT3306_BonChua2", out1 => "AI_TT3306_BonChua2_Eff")
   END_RUNG
   // the same network as SCL:
   IF NOT "AI_TT3306_BonChua2_Sim_Active" THEN "AI_TT3306_BonChua2_Eff" := "AI_TT3306_BonChua2"; END_IF;
END_REGION

REGION Network 25: Yêu cầu mô phỏng AI_PI3308_Truoc_Filter từ HMI
   RUNG wire#powerrail
      Contact( "AI_HMI_Use_Sim_Input_BonChua" )
      wire#w1
      Coil( "AI_PI3308_Truoc_Filter_Sim_Req" )
   END_RUNG
   RUNG wire#powerrail
      Contact( "AI_PI3308_Truoc_Filter_Use_HMI" )
   END_RUNG wire#w1
   // the same network as SCL:
   "AI_PI3308_Truoc_Filter_Sim_Req" := "AI_HMI_Use_Sim_Input_BonChua" OR "AI_PI3308_Truoc_Filter_Use_HMI";
END_REGION

REGION Network 26: Kích hoạt mô phỏng AI_PI3308_Truoc_Filter khi ở chế độ Sim Mode
   RUNG wire#powerrail
      Contact( "AI_HMI_Sim_Mode" )
      Contact( "AI_PI3308_Truoc_Filter_Sim_Req" )
      Coil( "AI_PI3308_Truoc_Filter_Sim_Active" )
   END_RUNG
   // the same network as SCL:
   "AI_PI3308_Truoc_Filter_Sim_Active" := "AI_HMI_Sim_Mode" AND "AI_PI3308_Truoc_Filter_Sim_Req";
END_REGION

REGION Network 27: Đọc giá trị mô phỏng AI_PI3308_Truoc_Filter vào hiệu dụng
   RUNG wire#powerrail
      Contact( "AI_PI3308_Truoc_Filter_Sim_Active" )
      { S7_GenerateENO := "TRUE" } Move(in := "AI_PI3308_Truoc_Filter_HMI", out1 => "AI_PI3308_Truoc_Filter_Eff")
   END_RUNG
   // the same network as SCL:
   IF "AI_PI3308_Truoc_Filter_Sim_Active" THEN
       "AI_PI3308_Truoc_Filter_Eff" := "AI_PI3308_Truoc_Filter_HMI";
   END_IF;
END_REGION

REGION Network 28: Đọc giá trị vật lý AI_PI3308_Truoc_Filter vào hiệu dụng
   RUNG wire#powerrail
      I_Contact( "AI_PI3308_Truoc_Filter_Sim_Active" )
      { S7_GenerateENO := "TRUE" } Move(in := "AI_PI3308_Truoc_Filter", out1 => "AI_PI3308_Truoc_Filter_Eff")
   END_RUNG
   // the same network as SCL:
   IF NOT "AI_PI3308_Truoc_Filter_Sim_Active" THEN
       "AI_PI3308_Truoc_Filter_Eff" := "AI_PI3308_Truoc_Filter";
   END_IF;
END_REGION

REGION Network 29: Yêu cầu mô phỏng AI_FT3309_Xa_Thanh_Pham từ HMI
   RUNG wire#powerrail
      Contact( "AI_HMI_Use_Sim_Input_BonChua" )
      wire#w1
      Coil( "AI_FT3309_Xa_Thanh_Pham_Sim_Req" )
   END_RUNG
   RUNG wire#powerrail
      Contact( "AI_FT3309_Xa_Thanh_Pham_Use_HMI" )
   END_RUNG wire#w1
   // the same network as SCL:
   "AI_FT3309_Xa_Thanh_Pham_Sim_Req" := "AI_HMI_Use_Sim_Input_BonChua" OR "AI_FT3309_Xa_Thanh_Pham_Use_HMI";
END_REGION

REGION Network 30: Kích hoạt mô phỏng AI_FT3309_Xa_Thanh_Pham khi ở chế độ Sim Mode
   RUNG wire#powerrail
      Contact( "AI_HMI_Sim_Mode" )
      Contact( "AI_FT3309_Xa_Thanh_Pham_Sim_Req" )
      Coil( "AI_FT3309_Xa_Thanh_Pham_Sim_Active" )
   END_RUNG
   // the same network as SCL:
   "AI_FT3309_Xa_Thanh_Pham_Sim_Active" := "AI_HMI_Sim_Mode" AND "AI_FT3309_Xa_Thanh_Pham_Sim_Req";
END_REGION

REGION Network 31: Đọc giá trị mô phỏng AI_FT3309_Xa_Thanh_Pham vào hiệu dụng
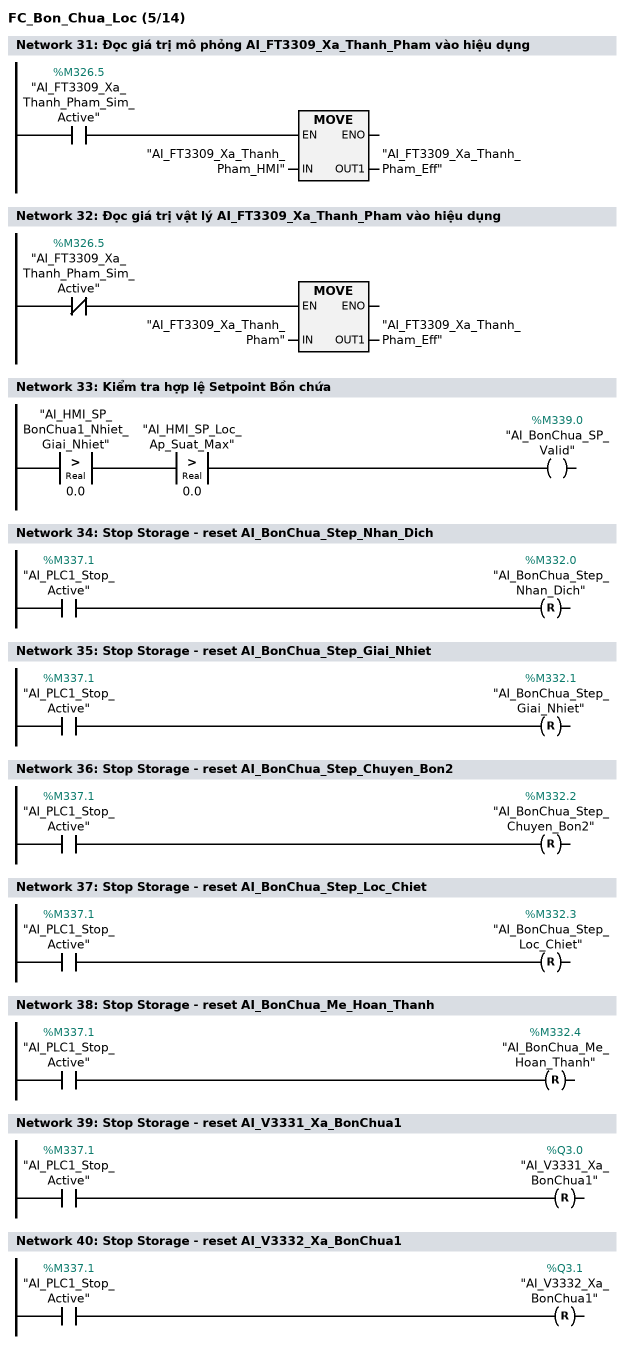
   RUNG wire#powerrail
      Contact( "AI_FT3309_Xa_Thanh_Pham_Sim_Active" )
      { S7_GenerateENO := "TRUE" } Move(in := "AI_FT3309_Xa_Thanh_Pham_HMI", out1 => "AI_FT3309_Xa_Thanh_Pham_Eff")
   END_RUNG
   // the same network as SCL:
   IF "AI_FT3309_Xa_Thanh_Pham_Sim_Active" THEN
       "AI_FT3309_Xa_Thanh_Pham_Eff" := "AI_FT3309_Xa_Thanh_Pham_HMI";
   END_IF;
END_REGION

REGION Network 32: Đọc giá trị vật lý AI_FT3309_Xa_Thanh_Pham vào hiệu dụng
   RUNG wire#powerrail
      I_Contact( "AI_FT3309_Xa_Thanh_Pham_Sim_Active" )
      { S7_GenerateENO := "TRUE" } Move(in := "AI_FT3309_Xa_Thanh_Pham", out1 => "AI_FT3309_Xa_Thanh_Pham_Eff")
   END_RUNG
   // the same network as SCL:
   IF NOT "AI_FT3309_Xa_Thanh_Pham_Sim_Active" THEN
       "AI_FT3309_Xa_Thanh_Pham_Eff" := "AI_FT3309_Xa_Thanh_Pham";
   END_IF;
END_REGION

REGION Network 33: Kiểm tra hợp lệ Setpoint Bồn chứa
   RUNG wire#powerrail
      { S7_Templates := "SrcType := Real" } GT_Contact(in1 := "AI_HMI_SP_BonChua1_Nhiet_Giai_Nhiet", in2 := 0.0)
      { S7_Templates := "SrcType := Real" } GT_Contact(in1 := "AI_HMI_SP_Loc_Ap_Suat_Max", in2 := 0.0)
      Coil( "AI_BonChua_SP_Valid" )
   END_RUNG
   // the same network as SCL:
   "AI_BonChua_SP_Valid" := ("AI_HMI_SP_BonChua1_Nhiet_Giai_Nhiet" > 0.0) AND ("AI_HMI_SP_Loc_Ap_Suat_Max" > 0.0);
END_REGION

REGION Network 34: Stop Storage - reset AI_BonChua_Step_Nhan_Dich
   RUNG wire#powerrail
      Contact( "AI_PLC1_Stop_Active" )
      R_Coil( "AI_BonChua_Step_Nhan_Dich" )
   END_RUNG
   // the same network as SCL:
   IF "AI_PLC1_Stop_Active" THEN "AI_BonChua_Step_Nhan_Dich" := FALSE; END_IF;
END_REGION

REGION Network 35: Stop Storage - reset AI_BonChua_Step_Giai_Nhiet
   RUNG wire#powerrail
      Contact( "AI_PLC1_Stop_Active" )
      R_Coil( "AI_BonChua_Step_Giai_Nhiet" )
   END_RUNG
   // the same network as SCL:
   IF "AI_PLC1_Stop_Active" THEN "AI_BonChua_Step_Giai_Nhiet" := FALSE; END_IF;
END_REGION

REGION Network 36: Stop Storage - reset AI_BonChua_Step_Chuyen_Bon2
   RUNG wire#powerrail
      Contact( "AI_PLC1_Stop_Active" )
      R_Coil( "AI_BonChua_Step_Chuyen_Bon2" )
   END_RUNG
   // the same network as SCL:
   IF "AI_PLC1_Stop_Active" THEN "AI_BonChua_Step_Chuyen_Bon2" := FALSE; END_IF;
END_REGION

REGION Network 37: Stop Storage - reset AI_BonChua_Step_Loc_Chiet
   RUNG wire#powerrail
      Contact( "AI_PLC1_Stop_Active" )
      R_Coil( "AI_BonChua_Step_Loc_Chiet" )
   END_RUNG
   // the same network as SCL:
   IF "AI_PLC1_Stop_Active" THEN "AI_BonChua_Step_Loc_Chiet" := FALSE; END_IF;
END_REGION

REGION Network 38: Stop Storage - reset AI_BonChua_Me_Hoan_Thanh
   RUNG wire#powerrail
      Contact( "AI_PLC1_Stop_Active" )
      R_Coil( "AI_BonChua_Me_Hoan_Thanh" )
   END_RUNG
   // the same network as SCL:
   IF "AI_PLC1_Stop_Active" THEN "AI_BonChua_Me_Hoan_Thanh" := FALSE; END_IF;
END_REGION

REGION Network 39: Stop Storage - reset AI_V3331_Xa_BonChua1
   RUNG wire#powerrail
      Contact( "AI_PLC1_Stop_Active" )
      R_Coil( "AI_V3331_Xa_BonChua1" )
   END_RUNG
   // the same network as SCL:
   IF "AI_PLC1_Stop_Active" THEN "AI_V3331_Xa_BonChua1" := FALSE; END_IF;
END_REGION

REGION Network 40: Stop Storage - reset AI_V3332_Xa_BonChua1
   RUNG wire#powerrail
      Contact( "AI_PLC1_Stop_Active" )
      R_Coil( "AI_V3332_Xa_BonChua1" )
   END_RUNG
   // the same network as SCL:
   IF "AI_PLC1_Stop_Active" THEN "AI_V3332_Xa_BonChua1" := FALSE; END_IF;
END_REGION

REGION Network 41: Stop Storage - reset AI_Pump3361_LuanChuyen_BonChua1
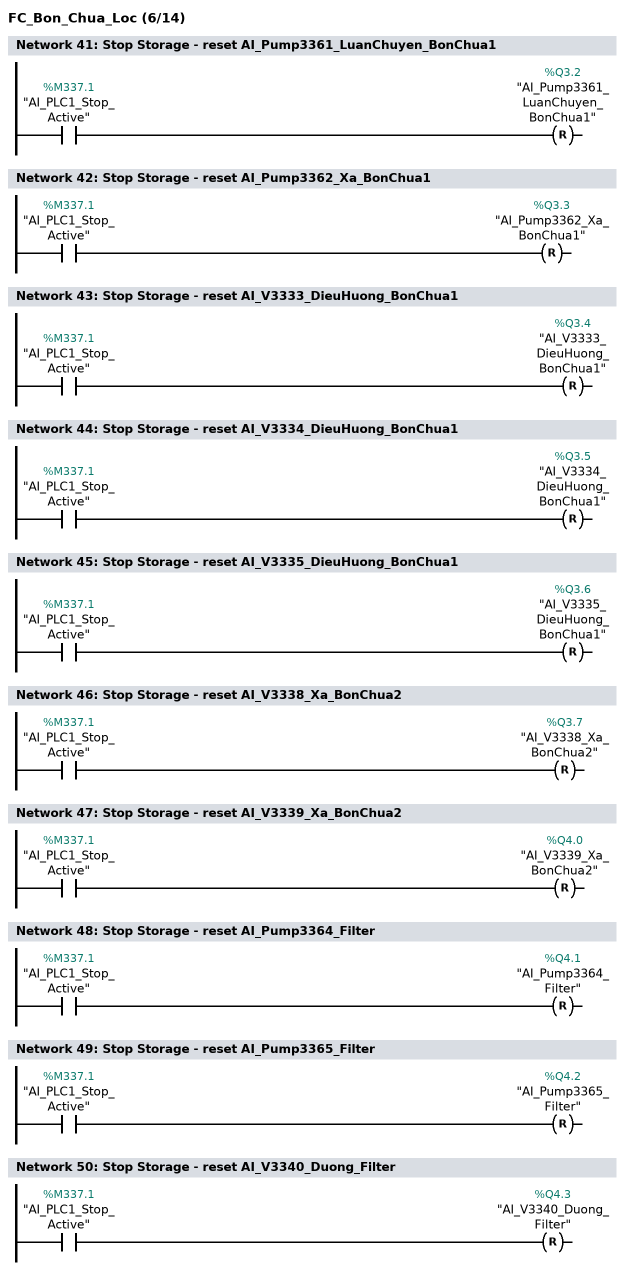
   RUNG wire#powerrail
      Contact( "AI_PLC1_Stop_Active" )
      R_Coil( "AI_Pump3361_LuanChuyen_BonChua1" )
   END_RUNG
   // the same network as SCL:
   IF "AI_PLC1_Stop_Active" THEN "AI_Pump3361_LuanChuyen_BonChua1" := FALSE; END_IF;
END_REGION

REGION Network 42: Stop Storage - reset AI_Pump3362_Xa_BonChua1
   RUNG wire#powerrail
      Contact( "AI_PLC1_Stop_Active" )
      R_Coil( "AI_Pump3362_Xa_BonChua1" )
   END_RUNG
   // the same network as SCL:
   IF "AI_PLC1_Stop_Active" THEN "AI_Pump3362_Xa_BonChua1" := FALSE; END_IF;
END_REGION

REGION Network 43: Stop Storage - reset AI_V3333_DieuHuong_BonChua1
   RUNG wire#powerrail
      Contact( "AI_PLC1_Stop_Active" )
      R_Coil( "AI_V3333_DieuHuong_BonChua1" )
   END_RUNG
   // the same network as SCL:
   IF "AI_PLC1_Stop_Active" THEN "AI_V3333_DieuHuong_BonChua1" := FALSE; END_IF;
END_REGION

REGION Network 44: Stop Storage - reset AI_V3334_DieuHuong_BonChua1
   RUNG wire#powerrail
      Contact( "AI_PLC1_Stop_Active" )
      R_Coil( "AI_V3334_DieuHuong_BonChua1" )
   END_RUNG
   // the same network as SCL:
   IF "AI_PLC1_Stop_Active" THEN "AI_V3334_DieuHuong_BonChua1" := FALSE; END_IF;
END_REGION

REGION Network 45: Stop Storage - reset AI_V3335_DieuHuong_BonChua1
   RUNG wire#powerrail
      Contact( "AI_PLC1_Stop_Active" )
      R_Coil( "AI_V3335_DieuHuong_BonChua1" )
   END_RUNG
   // the same network as SCL:
   IF "AI_PLC1_Stop_Active" THEN "AI_V3335_DieuHuong_BonChua1" := FALSE; END_IF;
END_REGION

REGION Network 46: Stop Storage - reset AI_V3338_Xa_BonChua2
   RUNG wire#powerrail
      Contact( "AI_PLC1_Stop_Active" )
      R_Coil( "AI_V3338_Xa_BonChua2" )
   END_RUNG
   // the same network as SCL:
   IF "AI_PLC1_Stop_Active" THEN "AI_V3338_Xa_BonChua2" := FALSE; END_IF;
END_REGION

REGION Network 47: Stop Storage - reset AI_V3339_Xa_BonChua2
   RUNG wire#powerrail
      Contact( "AI_PLC1_Stop_Active" )
      R_Coil( "AI_V3339_Xa_BonChua2" )
   END_RUNG
   // the same network as SCL:
   IF "AI_PLC1_Stop_Active" THEN "AI_V3339_Xa_BonChua2" := FALSE; END_IF;
END_REGION

REGION Network 48: Stop Storage - reset AI_Pump3364_Filter
   RUNG wire#powerrail
      Contact( "AI_PLC1_Stop_Active" )
      R_Coil( "AI_Pump3364_Filter" )
   END_RUNG
   // the same network as SCL:
   IF "AI_PLC1_Stop_Active" THEN "AI_Pump3364_Filter" := FALSE; END_IF;
END_REGION

REGION Network 49: Stop Storage - reset AI_Pump3365_Filter
   RUNG wire#powerrail
      Contact( "AI_PLC1_Stop_Active" )
      R_Coil( "AI_Pump3365_Filter" )
   END_RUNG
   // the same network as SCL:
   IF "AI_PLC1_Stop_Active" THEN "AI_Pump3365_Filter" := FALSE; END_IF;
END_REGION

REGION Network 50: Stop Storage - reset AI_V3340_Duong_Filter
   RUNG wire#powerrail
      Contact( "AI_PLC1_Stop_Active" )
      R_Coil( "AI_V3340_Duong_Filter" )
   END_RUNG
   // the same network as SCL:
   IF "AI_PLC1_Stop_Active" THEN "AI_V3340_Duong_Filter" := FALSE; END_IF;
END_REGION

REGION Network 51: Stop Storage - reset AI_V3341_Duong_Filter
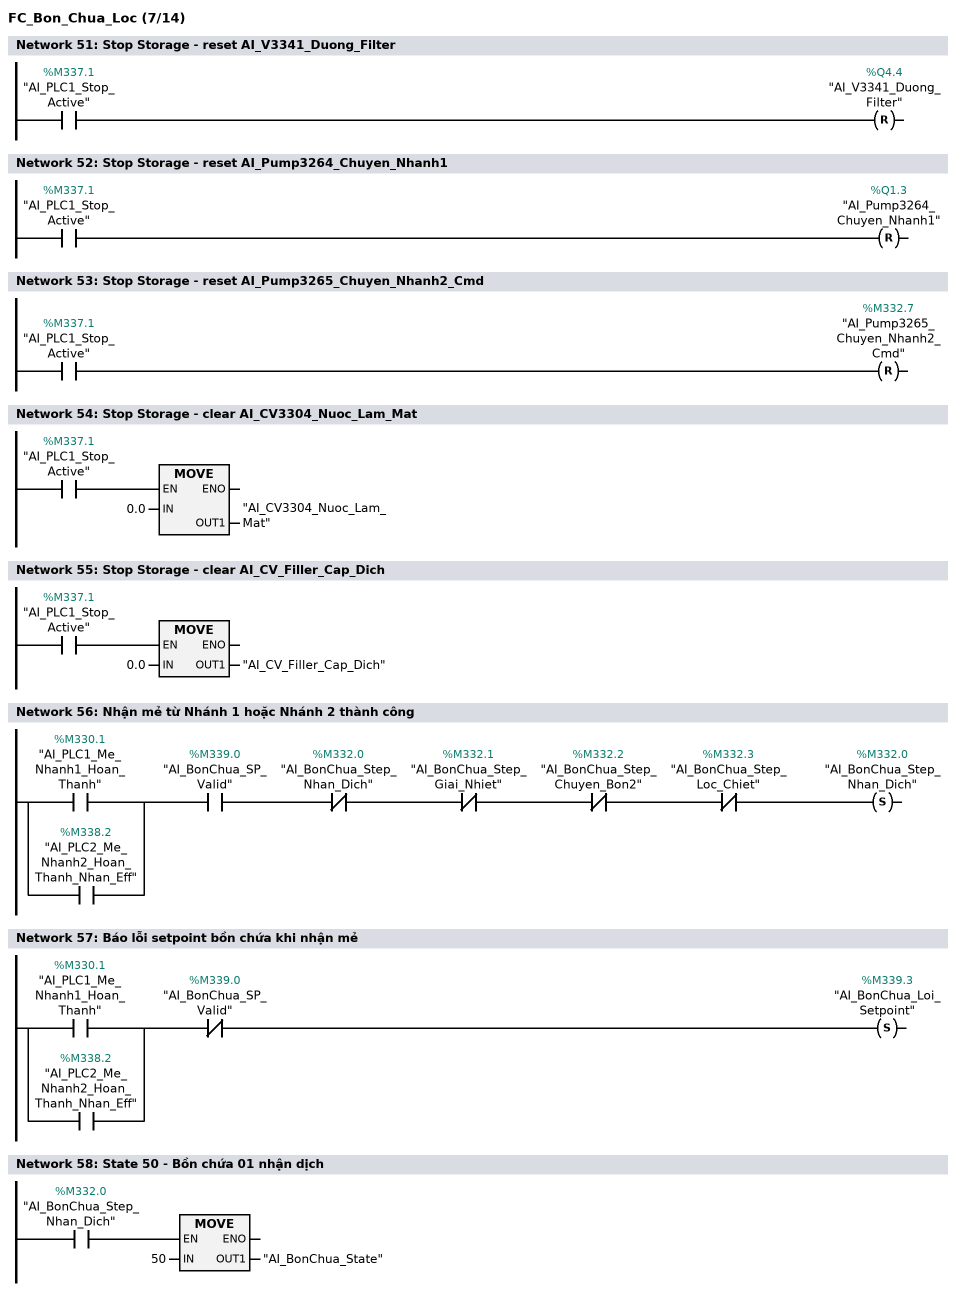
   RUNG wire#powerrail
      Contact( "AI_PLC1_Stop_Active" )
      R_Coil( "AI_V3341_Duong_Filter" )
   END_RUNG
   // the same network as SCL:
   IF "AI_PLC1_Stop_Active" THEN "AI_V3341_Duong_Filter" := FALSE; END_IF;
END_REGION

REGION Network 52: Stop Storage - reset AI_Pump3264_Chuyen_Nhanh1
   RUNG wire#powerrail
      Contact( "AI_PLC1_Stop_Active" )
      R_Coil( "AI_Pump3264_Chuyen_Nhanh1" )
   END_RUNG
   // the same network as SCL:
   IF "AI_PLC1_Stop_Active" THEN "AI_Pump3264_Chuyen_Nhanh1" := FALSE; END_IF;
END_REGION

REGION Network 53: Stop Storage - reset AI_Pump3265_Chuyen_Nhanh2_Cmd
   RUNG wire#powerrail
      Contact( "AI_PLC1_Stop_Active" )
      R_Coil( "AI_Pump3265_Chuyen_Nhanh2_Cmd" )
   END_RUNG
   // the same network as SCL:
   IF "AI_PLC1_Stop_Active" THEN "AI_Pump3265_Chuyen_Nhanh2_Cmd" := FALSE; END_IF;
END_REGION

REGION Network 54: Stop Storage - clear AI_CV3304_Nuoc_Lam_Mat
   RUNG wire#powerrail
      Contact( "AI_PLC1_Stop_Active" )
      { S7_GenerateENO := "TRUE" } Move(in := 0.0, out1 => "AI_CV3304_Nuoc_Lam_Mat")
   END_RUNG
   // the same network as SCL:
   IF "AI_PLC1_Stop_Active" THEN "AI_CV3304_Nuoc_Lam_Mat" := 0.0; END_IF;
END_REGION

REGION Network 55: Stop Storage - clear AI_CV_Filler_Cap_Dich
   RUNG wire#powerrail
      Contact( "AI_PLC1_Stop_Active" )
      { S7_GenerateENO := "TRUE" } Move(in := 0.0, out1 => "AI_CV_Filler_Cap_Dich")
   END_RUNG
   // the same network as SCL:
   IF "AI_PLC1_Stop_Active" THEN "AI_CV_Filler_Cap_Dich" := 0.0; END_IF;
END_REGION

REGION Network 56: Nhận mẻ từ Nhánh 1 hoặc Nhánh 2 thành công
   RUNG wire#powerrail
      Contact( "AI_PLC1_Me_Nhanh1_Hoan_Thanh" )
      wire#w1
      Contact( "AI_BonChua_SP_Valid" )
      I_Contact( "AI_BonChua_Step_Nhan_Dich" )
      I_Contact( "AI_BonChua_Step_Giai_Nhiet" )
      I_Contact( "AI_BonChua_Step_Chuyen_Bon2" )
      I_Contact( "AI_BonChua_Step_Loc_Chiet" )
      S_Coil( "AI_BonChua_Step_Nhan_Dich" )
   END_RUNG
   RUNG wire#powerrail
      Contact( "AI_PLC2_Me_Nhanh2_Hoan_Thanh_Nhan_Eff" )
   END_RUNG wire#w1
   // the same network as SCL:
   IF ("AI_PLC1_Me_Nhanh1_Hoan_Thanh" OR "AI_PLC2_Me_Nhanh2_Hoan_Thanh_Nhan_Eff") AND "AI_BonChua_SP_Valid" AND NOT "AI_BonChua_Step_Nhan_Dich" AND NOT "AI_BonChua_Step_Giai_Nhiet" AND NOT "AI_BonChua_Step_Chuyen_Bon2" AND NOT "AI_BonChua_Step_Loc_Chiet" THEN
       "AI_BonChua_Step_Nhan_Dich" := TRUE;
   END_IF;
END_REGION

REGION Network 57: Báo lỗi setpoint bồn chứa khi nhận mẻ
   RUNG wire#powerrail
      Contact( "AI_PLC1_Me_Nhanh1_Hoan_Thanh" )
      wire#w1
      I_Contact( "AI_BonChua_SP_Valid" )
      S_Coil( "AI_BonChua_Loi_Setpoint" )
   END_RUNG
   RUNG wire#powerrail
      Contact( "AI_PLC2_Me_Nhanh2_Hoan_Thanh_Nhan_Eff" )
   END_RUNG wire#w1
   // the same network as SCL:
   IF ("AI_PLC1_Me_Nhanh1_Hoan_Thanh" OR "AI_PLC2_Me_Nhanh2_Hoan_Thanh_Nhan_Eff") AND NOT "AI_BonChua_SP_Valid" THEN
       "AI_BonChua_Loi_Setpoint" := TRUE;
   END_IF;
END_REGION

REGION Network 58: State 50 - Bồn chứa 01 nhận dịch
   RUNG wire#powerrail
      Contact( "AI_BonChua_Step_Nhan_Dich" )
      { S7_GenerateENO := "TRUE" } Move(in := 50, out1 => "AI_BonChua_State")
   END_RUNG
   // the same network as SCL:
   IF "AI_BonChua_Step_Nhan_Dich" THEN "AI_BonChua_State" := 50; END_IF;
END_REGION

REGION Network 59: Reset cờ hoàn thành mẻ khi bắt đầu nhận dịch mới
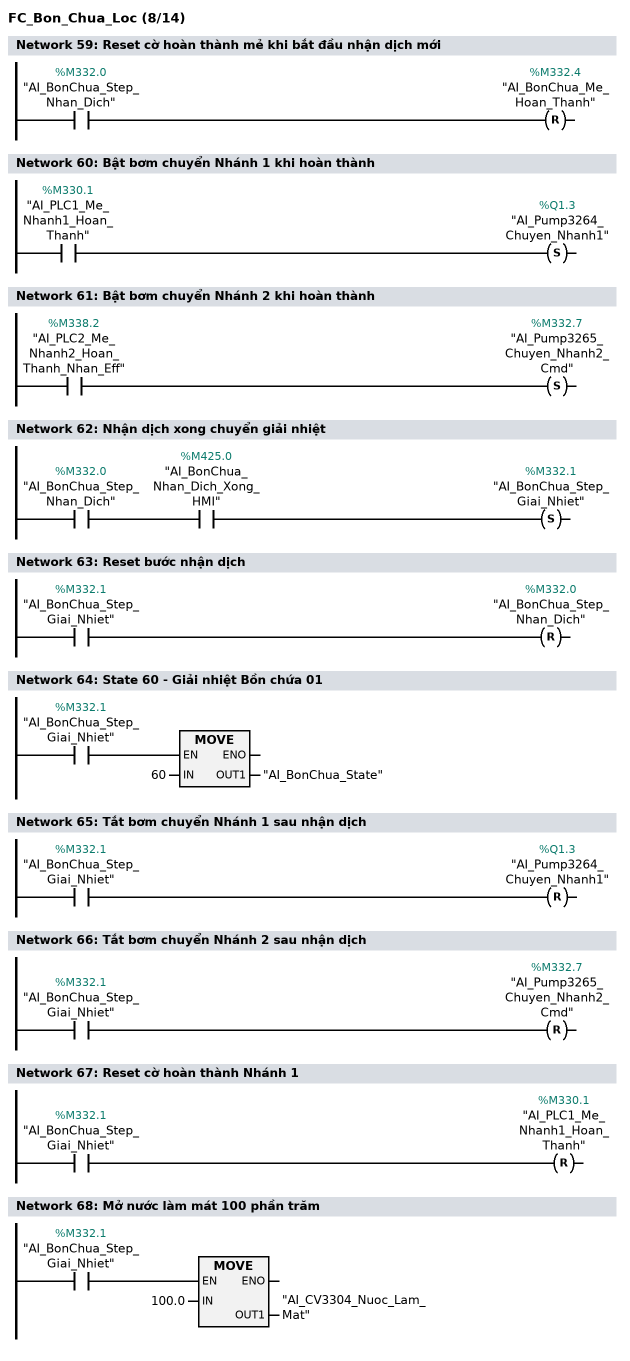
   RUNG wire#powerrail
      Contact( "AI_BonChua_Step_Nhan_Dich" )
      R_Coil( "AI_BonChua_Me_Hoan_Thanh" )
   END_RUNG
   // the same network as SCL:
   IF "AI_BonChua_Step_Nhan_Dich" THEN "AI_BonChua_Me_Hoan_Thanh" := FALSE; END_IF;
END_REGION

REGION Network 60: Bật bơm chuyển Nhánh 1 khi hoàn thành
   RUNG wire#powerrail
      Contact( "AI_PLC1_Me_Nhanh1_Hoan_Thanh" )
      S_Coil( "AI_Pump3264_Chuyen_Nhanh1" )
   END_RUNG
   // the same network as SCL:
   IF "AI_PLC1_Me_Nhanh1_Hoan_Thanh" THEN "AI_Pump3264_Chuyen_Nhanh1" := TRUE; END_IF;
END_REGION

REGION Network 61: Bật bơm chuyển Nhánh 2 khi hoàn thành
   RUNG wire#powerrail
      Contact( "AI_PLC2_Me_Nhanh2_Hoan_Thanh_Nhan_Eff" )
      S_Coil( "AI_Pump3265_Chuyen_Nhanh2_Cmd" )
   END_RUNG
   // the same network as SCL:
   IF "AI_PLC2_Me_Nhanh2_Hoan_Thanh_Nhan_Eff" THEN "AI_Pump3265_Chuyen_Nhanh2_Cmd" := TRUE; END_IF;
END_REGION

REGION Network 62: Nhận dịch xong chuyển giải nhiệt
   RUNG wire#powerrail
      Contact( "AI_BonChua_Step_Nhan_Dich" )
      Contact( "AI_BonChua_Nhan_Dich_Xong_HMI" )
      S_Coil( "AI_BonChua_Step_Giai_Nhiet" )
   END_RUNG
   // the same network as SCL:
   IF "AI_BonChua_Step_Nhan_Dich" AND "AI_BonChua_Nhan_Dich_Xong_HMI" THEN
       "AI_BonChua_Step_Giai_Nhiet" := TRUE;
   END_IF;
END_REGION

REGION Network 63: Reset bước nhận dịch
   RUNG wire#powerrail
      Contact( "AI_BonChua_Step_Giai_Nhiet" )
      R_Coil( "AI_BonChua_Step_Nhan_Dich" )
   END_RUNG
   // the same network as SCL:
   IF "AI_BonChua_Step_Giai_Nhiet" THEN "AI_BonChua_Step_Nhan_Dich" := FALSE; END_IF;
END_REGION

REGION Network 64: State 60 - Giải nhiệt Bồn chứa 01
   RUNG wire#powerrail
      Contact( "AI_BonChua_Step_Giai_Nhiet" )
      { S7_GenerateENO := "TRUE" } Move(in := 60, out1 => "AI_BonChua_State")
   END_RUNG
   // the same network as SCL:
   IF "AI_BonChua_Step_Giai_Nhiet" THEN "AI_BonChua_State" := 60; END_IF;
END_REGION

REGION Network 65: Tắt bơm chuyển Nhánh 1 sau nhận dịch
   RUNG wire#powerrail
      Contact( "AI_BonChua_Step_Giai_Nhiet" )
      R_Coil( "AI_Pump3264_Chuyen_Nhanh1" )
   END_RUNG
   // the same network as SCL:
   IF "AI_BonChua_Step_Giai_Nhiet" THEN "AI_Pump3264_Chuyen_Nhanh1" := FALSE; END_IF;
END_REGION

REGION Network 66: Tắt bơm chuyển Nhánh 2 sau nhận dịch
   RUNG wire#powerrail
      Contact( "AI_BonChua_Step_Giai_Nhiet" )
      R_Coil( "AI_Pump3265_Chuyen_Nhanh2_Cmd" )
   END_RUNG
   // the same network as SCL:
   IF "AI_BonChua_Step_Giai_Nhiet" THEN "AI_Pump3265_Chuyen_Nhanh2_Cmd" := FALSE; END_IF;
END_REGION

REGION Network 67: Reset cờ hoàn thành Nhánh 1
   RUNG wire#powerrail
      Contact( "AI_BonChua_Step_Giai_Nhiet" )
      R_Coil( "AI_PLC1_Me_Nhanh1_Hoan_Thanh" )
   END_RUNG
   // the same network as SCL:
   IF "AI_BonChua_Step_Giai_Nhiet" THEN "AI_PLC1_Me_Nhanh1_Hoan_Thanh" := FALSE; END_IF;
END_REGION

REGION Network 68: Mở nước làm mát 100 phần trăm
   RUNG wire#powerrail
      Contact( "AI_BonChua_Step_Giai_Nhiet" )
      { S7_GenerateENO := "TRUE" } Move(in := 100.0, out1 => "AI_CV3304_Nuoc_Lam_Mat")
   END_RUNG
   // the same network as SCL:
   IF "AI_BonChua_Step_Giai_Nhiet" THEN "AI_CV3304_Nuoc_Lam_Mat" := 100.0; END_IF;
END_REGION

REGION Network 69: Mở van xả đáy 01 để luân chuyển giải nhiệt
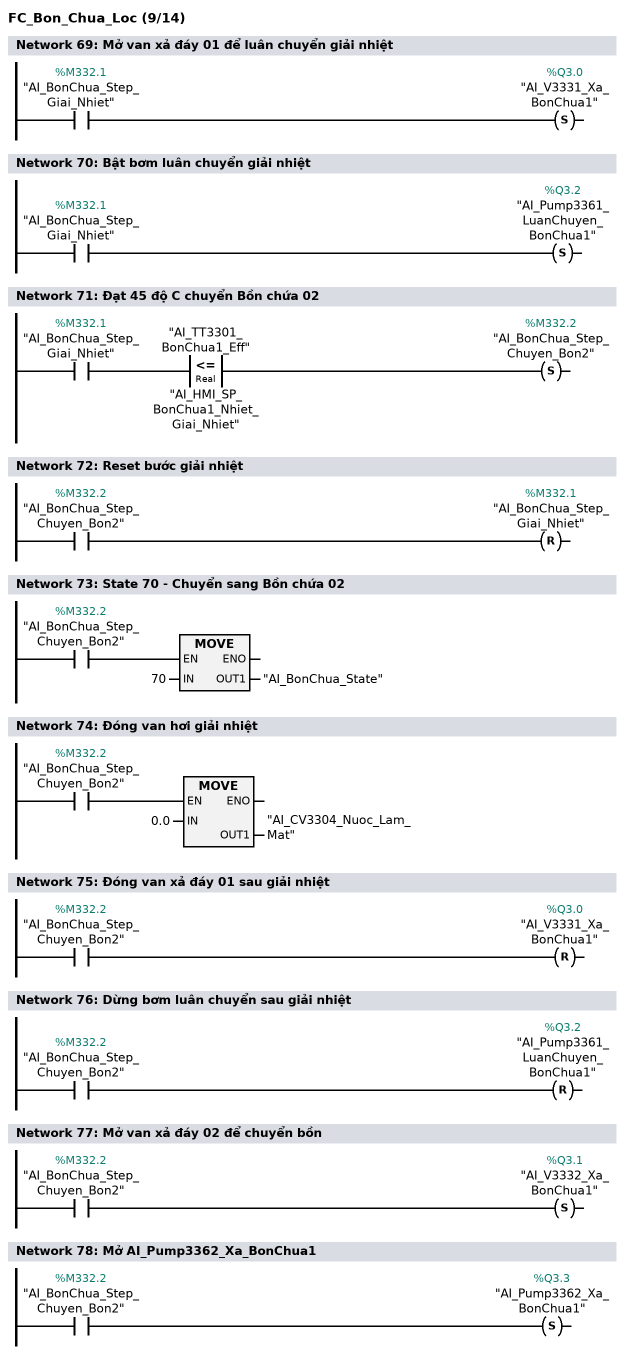
   RUNG wire#powerrail
      Contact( "AI_BonChua_Step_Giai_Nhiet" )
      S_Coil( "AI_V3331_Xa_BonChua1" )
   END_RUNG
   // the same network as SCL:
   IF "AI_BonChua_Step_Giai_Nhiet" THEN "AI_V3331_Xa_BonChua1" := TRUE; END_IF;
END_REGION

REGION Network 70: Bật bơm luân chuyển giải nhiệt
   RUNG wire#powerrail
      Contact( "AI_BonChua_Step_Giai_Nhiet" )
      S_Coil( "AI_Pump3361_LuanChuyen_BonChua1" )
   END_RUNG
   // the same network as SCL:
   IF "AI_BonChua_Step_Giai_Nhiet" THEN "AI_Pump3361_LuanChuyen_BonChua1" := TRUE; END_IF;
END_REGION

REGION Network 71: Đạt 45 độ C chuyển Bồn chứa 02
   RUNG wire#powerrail
      Contact( "AI_BonChua_Step_Giai_Nhiet" )
      { S7_Templates := "SrcType := Real" } LE_Contact(in1 := "AI_TT3301_BonChua1_Eff", in2 := "AI_HMI_SP_BonChua1_Nhiet_Giai_Nhiet")
      S_Coil( "AI_BonChua_Step_Chuyen_Bon2" )
   END_RUNG
   // the same network as SCL:
   IF "AI_BonChua_Step_Giai_Nhiet" AND ("AI_TT3301_BonChua1_Eff" <= "AI_HMI_SP_BonChua1_Nhiet_Giai_Nhiet") THEN
       "AI_BonChua_Step_Chuyen_Bon2" := TRUE;
   END_IF;
END_REGION

REGION Network 72: Reset bước giải nhiệt
   RUNG wire#powerrail
      Contact( "AI_BonChua_Step_Chuyen_Bon2" )
      R_Coil( "AI_BonChua_Step_Giai_Nhiet" )
   END_RUNG
   // the same network as SCL:
   IF "AI_BonChua_Step_Chuyen_Bon2" THEN "AI_BonChua_Step_Giai_Nhiet" := FALSE; END_IF;
END_REGION

REGION Network 73: State 70 - Chuyển sang Bồn chứa 02
   RUNG wire#powerrail
      Contact( "AI_BonChua_Step_Chuyen_Bon2" )
      { S7_GenerateENO := "TRUE" } Move(in := 70, out1 => "AI_BonChua_State")
   END_RUNG
   // the same network as SCL:
   IF "AI_BonChua_Step_Chuyen_Bon2" THEN "AI_BonChua_State" := 70; END_IF;
END_REGION

REGION Network 74: Đóng van hơi giải nhiệt
   RUNG wire#powerrail
      Contact( "AI_BonChua_Step_Chuyen_Bon2" )
      { S7_GenerateENO := "TRUE" } Move(in := 0.0, out1 => "AI_CV3304_Nuoc_Lam_Mat")
   END_RUNG
   // the same network as SCL:
   IF "AI_BonChua_Step_Chuyen_Bon2" THEN "AI_CV3304_Nuoc_Lam_Mat" := 0.0; END_IF;
END_REGION

REGION Network 75: Đóng van xả đáy 01 sau giải nhiệt
   RUNG wire#powerrail
      Contact( "AI_BonChua_Step_Chuyen_Bon2" )
      R_Coil( "AI_V3331_Xa_BonChua1" )
   END_RUNG
   // the same network as SCL:
   IF "AI_BonChua_Step_Chuyen_Bon2" THEN "AI_V3331_Xa_BonChua1" := FALSE; END_IF;
END_REGION

REGION Network 76: Dừng bơm luân chuyển sau giải nhiệt
   RUNG wire#powerrail
      Contact( "AI_BonChua_Step_Chuyen_Bon2" )
      R_Coil( "AI_Pump3361_LuanChuyen_BonChua1" )
   END_RUNG
   // the same network as SCL:
   IF "AI_BonChua_Step_Chuyen_Bon2" THEN "AI_Pump3361_LuanChuyen_BonChua1" := FALSE; END_IF;
END_REGION

REGION Network 77: Mở van xả đáy 02 để chuyển bồn
   RUNG wire#powerrail
      Contact( "AI_BonChua_Step_Chuyen_Bon2" )
      S_Coil( "AI_V3332_Xa_BonChua1" )
   END_RUNG
   // the same network as SCL:
   IF "AI_BonChua_Step_Chuyen_Bon2" THEN "AI_V3332_Xa_BonChua1" := TRUE; END_IF;
END_REGION

REGION Network 78: Mở AI_Pump3362_Xa_BonChua1
   RUNG wire#powerrail
      Contact( "AI_BonChua_Step_Chuyen_Bon2" )
      S_Coil( "AI_Pump3362_Xa_BonChua1" )
   END_RUNG
   // the same network as SCL:
   IF "AI_BonChua_Step_Chuyen_Bon2" THEN "AI_Pump3362_Xa_BonChua1" := TRUE; END_IF;
END_REGION

REGION Network 79: Mở AI_V3333_DieuHuong_BonChua1
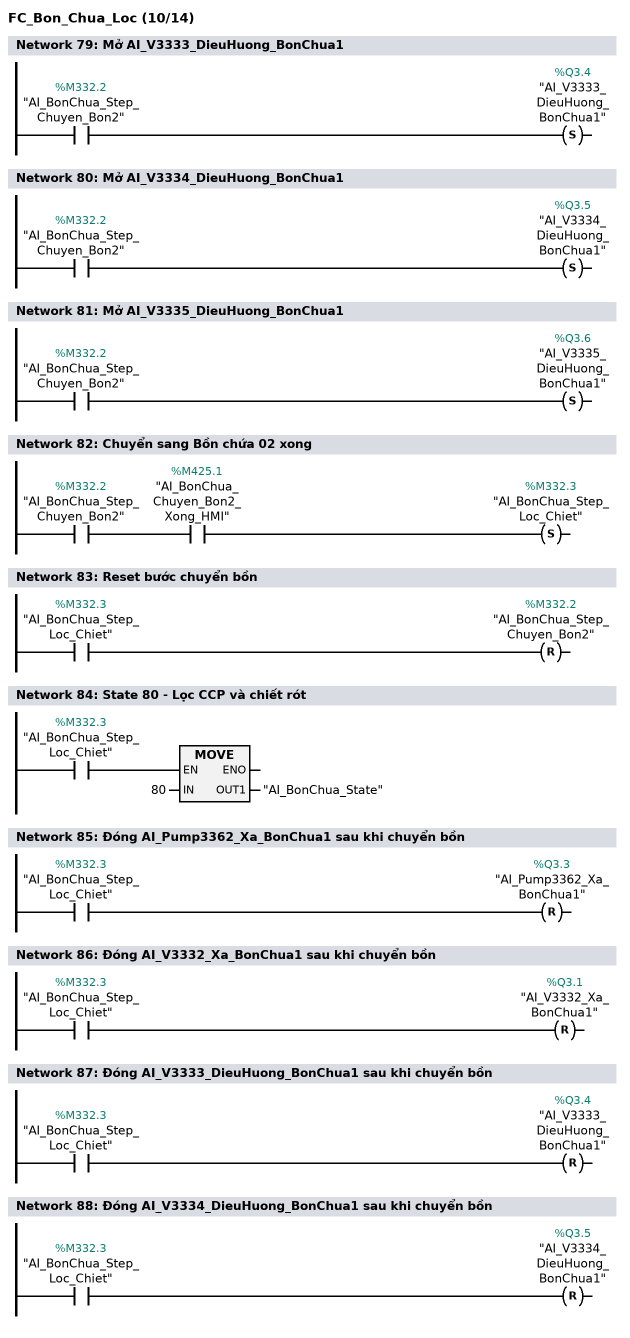
   RUNG wire#powerrail
      Contact( "AI_BonChua_Step_Chuyen_Bon2" )
      S_Coil( "AI_V3333_DieuHuong_BonChua1" )
   END_RUNG
   // the same network as SCL:
   IF "AI_BonChua_Step_Chuyen_Bon2" THEN "AI_V3333_DieuHuong_BonChua1" := TRUE; END_IF;
END_REGION

REGION Network 80: Mở AI_V3334_DieuHuong_BonChua1
   RUNG wire#powerrail
      Contact( "AI_BonChua_Step_Chuyen_Bon2" )
      S_Coil( "AI_V3334_DieuHuong_BonChua1" )
   END_RUNG
   // the same network as SCL:
   IF "AI_BonChua_Step_Chuyen_Bon2" THEN "AI_V3334_DieuHuong_BonChua1" := TRUE; END_IF;
END_REGION

REGION Network 81: Mở AI_V3335_DieuHuong_BonChua1
   RUNG wire#powerrail
      Contact( "AI_BonChua_Step_Chuyen_Bon2" )
      S_Coil( "AI_V3335_DieuHuong_BonChua1" )
   END_RUNG
   // the same network as SCL:
   IF "AI_BonChua_Step_Chuyen_Bon2" THEN "AI_V3335_DieuHuong_BonChua1" := TRUE; END_IF;
END_REGION

REGION Network 82: Chuyển sang Bồn chứa 02 xong
   RUNG wire#powerrail
      Contact( "AI_BonChua_Step_Chuyen_Bon2" )
      Contact( "AI_BonChua_Chuyen_Bon2_Xong_HMI" )
      S_Coil( "AI_BonChua_Step_Loc_Chiet" )
   END_RUNG
   // the same network as SCL:
   IF "AI_BonChua_Step_Chuyen_Bon2" AND "AI_BonChua_Chuyen_Bon2_Xong_HMI" THEN
       "AI_BonChua_Step_Loc_Chiet" := TRUE;
   END_IF;
END_REGION

REGION Network 83: Reset bước chuyển bồn
   RUNG wire#powerrail
      Contact( "AI_BonChua_Step_Loc_Chiet" )
      R_Coil( "AI_BonChua_Step_Chuyen_Bon2" )
   END_RUNG
   // the same network as SCL:
   IF "AI_BonChua_Step_Loc_Chiet" THEN "AI_BonChua_Step_Chuyen_Bon2" := FALSE; END_IF;
END_REGION

REGION Network 84: State 80 - Lọc CCP và chiết rót
   RUNG wire#powerrail
      Contact( "AI_BonChua_Step_Loc_Chiet" )
      { S7_GenerateENO := "TRUE" } Move(in := 80, out1 => "AI_BonChua_State")
   END_RUNG
   // the same network as SCL:
   IF "AI_BonChua_Step_Loc_Chiet" THEN "AI_BonChua_State" := 80; END_IF;
END_REGION

REGION Network 85: Đóng AI_Pump3362_Xa_BonChua1 sau khi chuyển bồn
   RUNG wire#powerrail
      Contact( "AI_BonChua_Step_Loc_Chiet" )
      R_Coil( "AI_Pump3362_Xa_BonChua1" )
   END_RUNG
   // the same network as SCL:
   IF "AI_BonChua_Step_Loc_Chiet" THEN "AI_Pump3362_Xa_BonChua1" := FALSE; END_IF;
END_REGION

REGION Network 86: Đóng AI_V3332_Xa_BonChua1 sau khi chuyển bồn
   RUNG wire#powerrail
      Contact( "AI_BonChua_Step_Loc_Chiet" )
      R_Coil( "AI_V3332_Xa_BonChua1" )
   END_RUNG
   // the same network as SCL:
   IF "AI_BonChua_Step_Loc_Chiet" THEN "AI_V3332_Xa_BonChua1" := FALSE; END_IF;
END_REGION

REGION Network 87: Đóng AI_V3333_DieuHuong_BonChua1 sau khi chuyển bồn
   RUNG wire#powerrail
      Contact( "AI_BonChua_Step_Loc_Chiet" )
      R_Coil( "AI_V3333_DieuHuong_BonChua1" )
   END_RUNG
   // the same network as SCL:
   IF "AI_BonChua_Step_Loc_Chiet" THEN "AI_V3333_DieuHuong_BonChua1" := FALSE; END_IF;
END_REGION

REGION Network 88: Đóng AI_V3334_DieuHuong_BonChua1 sau khi chuyển bồn
   RUNG wire#powerrail
      Contact( "AI_BonChua_Step_Loc_Chiet" )
      R_Coil( "AI_V3334_DieuHuong_BonChua1" )
   END_RUNG
   // the same network as SCL:
   IF "AI_BonChua_Step_Loc_Chiet" THEN "AI_V3334_DieuHuong_BonChua1" := FALSE; END_IF;
END_REGION

REGION Network 89: Đóng AI_V3335_DieuHuong_BonChua1 sau khi chuyển bồn
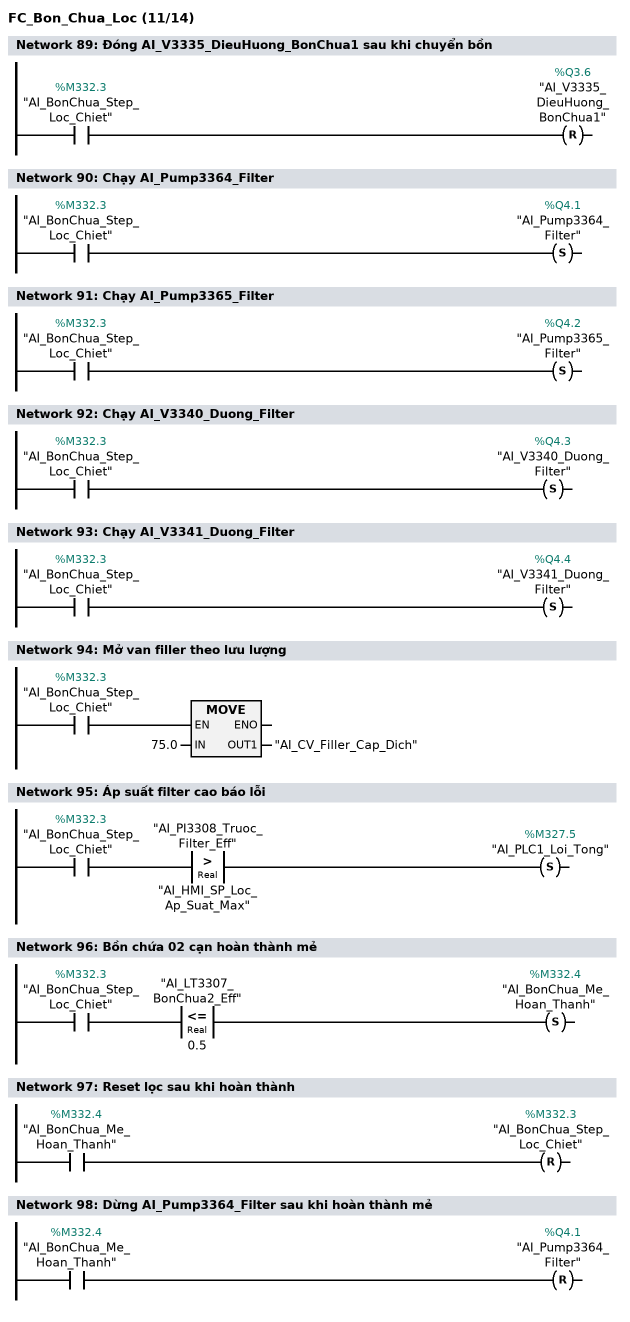
   RUNG wire#powerrail
      Contact( "AI_BonChua_Step_Loc_Chiet" )
      R_Coil( "AI_V3335_DieuHuong_BonChua1" )
   END_RUNG
   // the same network as SCL:
   IF "AI_BonChua_Step_Loc_Chiet" THEN "AI_V3335_DieuHuong_BonChua1" := FALSE; END_IF;
END_REGION

REGION Network 90: Chạy AI_Pump3364_Filter
   RUNG wire#powerrail
      Contact( "AI_BonChua_Step_Loc_Chiet" )
      S_Coil( "AI_Pump3364_Filter" )
   END_RUNG
   // the same network as SCL:
   IF "AI_BonChua_Step_Loc_Chiet" THEN "AI_Pump3364_Filter" := TRUE; END_IF;
END_REGION

REGION Network 91: Chạy AI_Pump3365_Filter
   RUNG wire#powerrail
      Contact( "AI_BonChua_Step_Loc_Chiet" )
      S_Coil( "AI_Pump3365_Filter" )
   END_RUNG
   // the same network as SCL:
   IF "AI_BonChua_Step_Loc_Chiet" THEN "AI_Pump3365_Filter" := TRUE; END_IF;
END_REGION

REGION Network 92: Chạy AI_V3340_Duong_Filter
   RUNG wire#powerrail
      Contact( "AI_BonChua_Step_Loc_Chiet" )
      S_Coil( "AI_V3340_Duong_Filter" )
   END_RUNG
   // the same network as SCL:
   IF "AI_BonChua_Step_Loc_Chiet" THEN "AI_V3340_Duong_Filter" := TRUE; END_IF;
END_REGION

REGION Network 93: Chạy AI_V3341_Duong_Filter
   RUNG wire#powerrail
      Contact( "AI_BonChua_Step_Loc_Chiet" )
      S_Coil( "AI_V3341_Duong_Filter" )
   END_RUNG
   // the same network as SCL:
   IF "AI_BonChua_Step_Loc_Chiet" THEN "AI_V3341_Duong_Filter" := TRUE; END_IF;
END_REGION

REGION Network 94: Mở van filler theo lưu lượng
   RUNG wire#powerrail
      Contact( "AI_BonChua_Step_Loc_Chiet" )
      { S7_GenerateENO := "TRUE" } Move(in := 75.0, out1 => "AI_CV_Filler_Cap_Dich")
   END_RUNG
   // the same network as SCL:
   IF "AI_BonChua_Step_Loc_Chiet" THEN "AI_CV_Filler_Cap_Dich" := 75.0; END_IF;
END_REGION

REGION Network 95: Áp suất filter cao báo lỗi
   RUNG wire#powerrail
      Contact( "AI_BonChua_Step_Loc_Chiet" )
      { S7_Templates := "SrcType := Real" } GT_Contact(in1 := "AI_PI3308_Truoc_Filter_Eff", in2 := "AI_HMI_SP_Loc_Ap_Suat_Max")
      S_Coil( "AI_PLC1_Loi_Tong" )
   END_RUNG
   // the same network as SCL:
   IF "AI_BonChua_Step_Loc_Chiet" AND ("AI_PI3308_Truoc_Filter_Eff" > "AI_HMI_SP_Loc_Ap_Suat_Max") THEN
       "AI_PLC1_Loi_Tong" := TRUE;
   END_IF;
END_REGION

REGION Network 96: Bồn chứa 02 cạn hoàn thành mẻ
   RUNG wire#powerrail
      Contact( "AI_BonChua_Step_Loc_Chiet" )
      { S7_Templates := "SrcType := Real" } LE_Contact(in1 := "AI_LT3307_BonChua2_Eff", in2 := 0.5)
      S_Coil( "AI_BonChua_Me_Hoan_Thanh" )
   END_RUNG
   // the same network as SCL:
   IF "AI_BonChua_Step_Loc_Chiet" AND ("AI_LT3307_BonChua2_Eff" <= 0.5) THEN
       "AI_BonChua_Me_Hoan_Thanh" := TRUE;
   END_IF;
END_REGION

REGION Network 97: Reset lọc sau khi hoàn thành
   RUNG wire#powerrail
      Contact( "AI_BonChua_Me_Hoan_Thanh" )
      R_Coil( "AI_BonChua_Step_Loc_Chiet" )
   END_RUNG
   // the same network as SCL:
   IF "AI_BonChua_Me_Hoan_Thanh" THEN "AI_BonChua_Step_Loc_Chiet" := FALSE; END_IF;
END_REGION

REGION Network 98: Dừng AI_Pump3364_Filter sau khi hoàn thành mẻ
   RUNG wire#powerrail
      Contact( "AI_BonChua_Me_Hoan_Thanh" )
      R_Coil( "AI_Pump3364_Filter" )
   END_RUNG
   // the same network as SCL:
   IF "AI_BonChua_Me_Hoan_Thanh" THEN "AI_Pump3364_Filter" := FALSE; END_IF;
END_REGION

REGION Network 99: Dừng AI_Pump3365_Filter sau khi hoàn thành mẻ
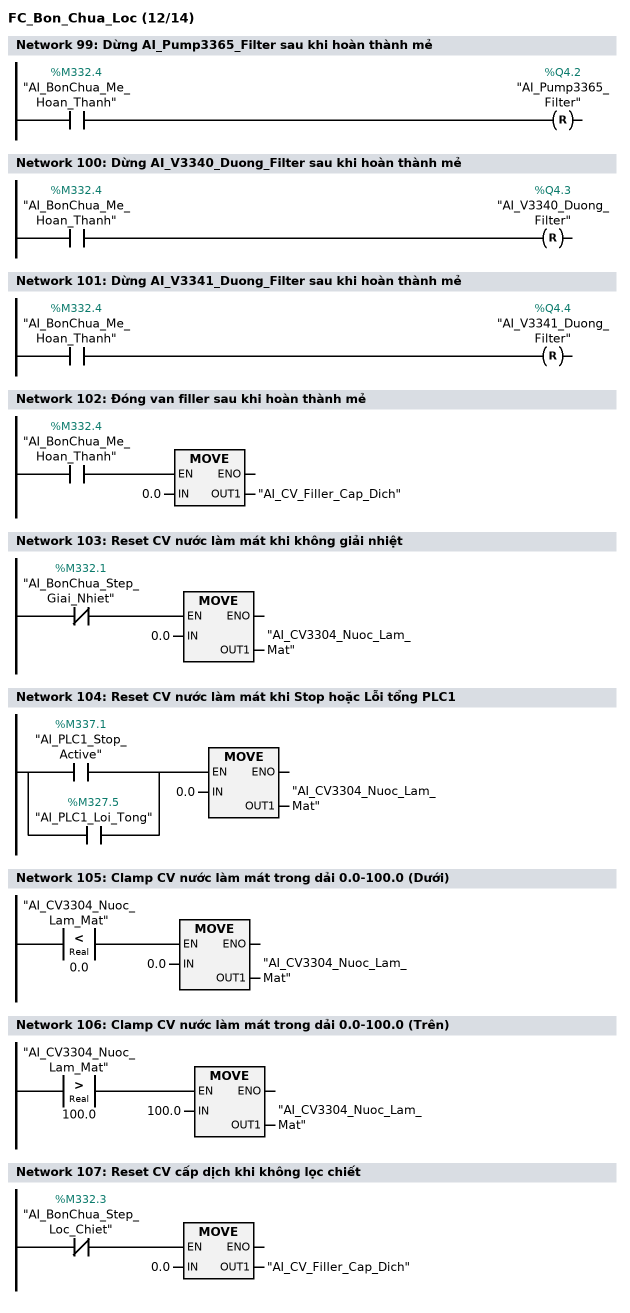
   RUNG wire#powerrail
      Contact( "AI_BonChua_Me_Hoan_Thanh" )
      R_Coil( "AI_Pump3365_Filter" )
   END_RUNG
   // the same network as SCL:
   IF "AI_BonChua_Me_Hoan_Thanh" THEN "AI_Pump3365_Filter" := FALSE; END_IF;
END_REGION

REGION Network 100: Dừng AI_V3340_Duong_Filter sau khi hoàn thành mẻ
   RUNG wire#powerrail
      Contact( "AI_BonChua_Me_Hoan_Thanh" )
      R_Coil( "AI_V3340_Duong_Filter" )
   END_RUNG
   // the same network as SCL:
   IF "AI_BonChua_Me_Hoan_Thanh" THEN "AI_V3340_Duong_Filter" := FALSE; END_IF;
END_REGION

REGION Network 101: Dừng AI_V3341_Duong_Filter sau khi hoàn thành mẻ
   RUNG wire#powerrail
      Contact( "AI_BonChua_Me_Hoan_Thanh" )
      R_Coil( "AI_V3341_Duong_Filter" )
   END_RUNG
   // the same network as SCL:
   IF "AI_BonChua_Me_Hoan_Thanh" THEN "AI_V3341_Duong_Filter" := FALSE; END_IF;
END_REGION

REGION Network 102: Đóng van filler sau khi hoàn thành mẻ
   RUNG wire#powerrail
      Contact( "AI_BonChua_Me_Hoan_Thanh" )
      { S7_GenerateENO := "TRUE" } Move(in := 0.0, out1 => "AI_CV_Filler_Cap_Dich")
   END_RUNG
   // the same network as SCL:
   IF "AI_BonChua_Me_Hoan_Thanh" THEN "AI_CV_Filler_Cap_Dich" := 0.0; END_IF;
END_REGION

REGION Network 103: Reset CV nước làm mát khi không giải nhiệt
   RUNG wire#powerrail
      I_Contact( "AI_BonChua_Step_Giai_Nhiet" )
      { S7_GenerateENO := "TRUE" } Move(in := 0.0, out1 => "AI_CV3304_Nuoc_Lam_Mat")
   END_RUNG
   // the same network as SCL:
   IF NOT "AI_BonChua_Step_Giai_Nhiet" THEN "AI_CV3304_Nuoc_Lam_Mat" := 0.0; END_IF;
END_REGION

REGION Network 104: Reset CV nước làm mát khi Stop hoặc Lỗi tổng PLC1
   RUNG wire#powerrail
      Contact( "AI_PLC1_Stop_Active" )
      wire#w1
      { S7_GenerateENO := "TRUE" } Move(in := 0.0, out1 => "AI_CV3304_Nuoc_Lam_Mat")
   END_RUNG
   RUNG wire#powerrail
      Contact( "AI_PLC1_Loi_Tong" )
   END_RUNG wire#w1
   // the same network as SCL:
   IF "AI_PLC1_Stop_Active" OR "AI_PLC1_Loi_Tong" THEN "AI_CV3304_Nuoc_Lam_Mat" := 0.0; END_IF;
END_REGION

REGION Network 105: Clamp CV nước làm mát trong dải 0.0-100.0 (Dưới)
   RUNG wire#powerrail
      { S7_Templates := "SrcType := Real" } LT_Contact(in1 := "AI_CV3304_Nuoc_Lam_Mat", in2 := 0.0)
      { S7_GenerateENO := "TRUE" } Move(in := 0.0, out1 => "AI_CV3304_Nuoc_Lam_Mat")
   END_RUNG
   // the same network as SCL:
   IF "AI_CV3304_Nuoc_Lam_Mat" < 0.0 THEN "AI_CV3304_Nuoc_Lam_Mat" := 0.0; END_IF;
END_REGION

REGION Network 106: Clamp CV nước làm mát trong dải 0.0-100.0 (Trên)
   RUNG wire#powerrail
      { S7_Templates := "SrcType := Real" } GT_Contact(in1 := "AI_CV3304_Nuoc_Lam_Mat", in2 := 100.0)
      { S7_GenerateENO := "TRUE" } Move(in := 100.0, out1 => "AI_CV3304_Nuoc_Lam_Mat")
   END_RUNG
   // the same network as SCL:
   IF "AI_CV3304_Nuoc_Lam_Mat" > 100.0 THEN "AI_CV3304_Nuoc_Lam_Mat" := 100.0; END_IF;
END_REGION

REGION Network 107: Reset CV cấp dịch khi không lọc chiết
   RUNG wire#powerrail
      I_Contact( "AI_BonChua_Step_Loc_Chiet" )
      { S7_GenerateENO := "TRUE" } Move(in := 0.0, out1 => "AI_CV_Filler_Cap_Dich")
   END_RUNG
   // the same network as SCL:
   IF NOT "AI_BonChua_Step_Loc_Chiet" THEN "AI_CV_Filler_Cap_Dich" := 0.0; END_IF;
END_REGION

REGION Network 108: Reset CV cấp dịch khi Stop hoặc Lỗi tổng PLC1
